LIN {X 0,Y 420.227,Z 348.89,A -85,B 0,C 180,E1 -10155.703,E2 -10155.703} C_VEL
LIN {X 0,Y 419.508,Z 359.488,A -85,B 0,C 180,E1 -10156.806,E2 -10156.806} C_VEL
LIN {X 0,Y 418.942,Z 368.019,A -85,B 0,C 180,E1 -10157.896,E2 -10157.896} C_VEL
LIN {X 0,Y 418.299,Z 375.888,A -85,B 0,C 180,E1 -10159.105,E2 -10159.105} C_VEL
LIN {X 0,Y 417.781,Z 383.575,A -85,B 0,C 180,E1 -10160.56,E2 -10160.56} C_VEL
LIN {X 0,Y 417.366,Z 390.664,A -85,B 0,C 180,E1 -10162.258,E2 -10162.258} C_VEL
LIN {X 0,Y 417.141,Z 395.456,A -85,B 0,C 180,E1 -10163.739,E2 -10163.739} C_VEL
LIN {X 0,Y 417.106,Z 398.985,A -85,B 0,C 180,E1 -10165.167,E2 -10165.167} C_VEL
LIN {X 0,Y 416.998,Z 400.842,A -85,B 0,C 180,E1 -10166.135,E2 -10166.135} C_VEL
LIN {X 0,Y 417.018,Z 402.236,A -85,B 0,C 180,E1 -10167.102,E2 -10167.102} C_VEL
LIN {X 0,Y 417.055,Z 403.232,A -85,B 0,C 180,E1 -10168.069,E2 -10168.069} C_VEL
LIN {X 0,Y 416.984,Z 404.052,A -85,B 0,C 180,E1 -10170,E2 -10170} C_VEL
LIN {X 0,Y 417.055,Z 403.229,A -85,B 0,C 180,E1 -10171.931,E2 -10171.931} C_VEL
LIN {X 0,Y 417.018,Z 402.232,A -85,B 0,C 180,E1 -10172.898,E2 -10172.898} C_VEL
LIN {X 0,Y 416.998,Z 400.835,A -85,B 0,C 180,E1 -10173.866,E2 -10173.866} C_VEL
LIN {X 0,Y 417.122,Z 397.902,A -85,B 0,C 180,E1 -10175.317,E2 -10175.317} C_VEL
LIN {X 0,Y 417.234,Z 393.93,A -85,B 0,C 180,E1 -10176.772,E2 -10176.772} C_VEL
LIN {X 0,Y 417.522,Z 387.822,A -85,B 0,C 180,E1 -10178.47,E2 -10178.47} C_VEL
LIN {X 0,Y 417.931,Z 381.149,A -85,B 0,C 180,E1 -10179.925,E2 -10179.925} C_VEL
LIN {X 0,Y 418.509,Z 372.87,A -85,B 0,C 180,E1 -10181.38,E2 -10181.38} C_VEL
LIN {X 0,Y 419.228,Z 364.386,A -85,B 0,C 180,E1 -10182.588,E2 -10182.588} C_VEL
LIN {X 0,Y 419.889,Z 353.882,A -85,B 0,C 180,E1 -10183.8,E2 -10183.8} C_VEL
LIN {X 0,Y 420.7,Z 342.093,A -85,B 0,C 180,E1 -10184.883,E2 -10184.883} C_VEL
LIN {X 0,Y 421.458,Z 330.219,A -85,B 0,C 180,E1 -10185.722,E2 -10185.722} C_VEL
LIN {X 0,Y 422.07,Z 317.862,A -85,B 0,C 180,E1 -10186.381,E2 -10186.381} C_VEL
LIN {X 0,Y 422.722,Z 305.172,A -85,B 0,C 180,E1 -10186.852,E2 -10186.852} C_VEL
LIN {X 0,Y 423.018,Z 291.859,A -85,B 0,C 180,E1 -10187.151,E2 -10187.151} C_VEL
LIN {X 0,Y 423.707,Z 215.963,A -85,B 0,C 180,E1 -10188.445,E2 -10188.445} C_VEL
LIN {X 0,Y 419.677,Z 191.543,A -85,B 0,C 180,E1 -10189.081,E2 -10189.081} C_VEL
LIN {X 0,Y 420.834,Z 174.196,A -85,B 0,C 180,E1 -10192.588,E2 -10192.588} C_VEL
LIN {X 0,Y 421.039,Z 167.944,A -85,B 0,C 180,E1 -10193.877,E2 -10193.877} C_VEL
LIN {X 0,Y 418.547,Z 155.355,A -85,B 0,C 180,E1 -10196.69,E2 -10196.69} C_VEL
LIN {X 0,Y 418.225,Z 153.888,A -85,B 0,C 180,E1 -10197.047,E2 -10197.047} C_VEL
LIN {X 0,Y 418.241,Z 153.882,A -85,B 0,C 180,E1 -10200.272,E2 -10200.272} C_VEL
LIN {X 0,Y 418.233,Z 153.885,A -85,B 0,C 180,E1 -10203.678,E2 -10203.678} C_VEL
LIN {X 0,Y 418.239,Z 153.886,A -85,B 0,C 180,E1 -10207.224,E2 -10207.224} C_VEL
LIN {X 0,Y 418.213,Z 153.892,A -85,B 0,C 180,E1 -10210.868,E2 -10210.868} C_VEL
LIN {X 0,Y 418.208,Z 153.887,A -85,B 0,C 180,E1 -10213.729,E2 -10213.729} C_VEL
LIN {X 0,Y 418.208,Z 153.894,A -85,B 0,C 180,E1 -10216.448,E2 -10216.448} C_VEL
LIN {X 0,Y 418.22,Z 153.886,A -85,B 0,C 180,E1 -10219.13,E2 -10219.13} C_VEL
LIN {X 0,Y 418.224,Z 153.89,A -85,B 0,C 180,E1 -10222.167,E2 -10222.167} C_VEL
LIN {X 0,Y 418.265,Z 153.88,A -85,B 0,C 180,E1 -10225.42,E2 -10225.42} C_VEL
LIN {X 0,Y 418.211,Z 153.889,A -85,B 0,C 180,E1 -10228.604,E2 -10228.604} C_VEL
LIN {X 0,Y 418.248,Z 153.888,A -85,B 0,C 180,E1 -10231.933,E2 -10231.933} C_VEL
LIN {X 0,Y 418.271,Z 153.88,A -85,B 0,C 180,E1 -10235.161,E2 -10235.161} C_VEL
LIN {X 0,Y 418.233,Z 153.887,A -85,B 0,C 180,E1 -10238.304,E2 -10238.304} C_VEL
LIN {X 0,Y 418.28,Z 153.881,A -85,B 0,C 180,E1 -10241.383,E2 -10241.383} C_VEL
LIN {X 0,Y 418.301,Z 153.876,A -85,B 0,C 180,E1 -10244.406,E2 -10244.406} C_VEL
LIN {X 0,Y 418.355,Z 153.873,A -85,B 0,C 180,E1 -10247.386,E2 -10247.386} C_VEL
LIN {X 0,Y 418.4,Z 153.868,A -85,B 0,C 180,E1 -10251.305,E2 -10251.305} C_VEL
LIN {X 0,Y 418.509,Z 153.85,A -85,B 0,C 180,E1 -10254.217,E2 -10254.217} C_VEL
LIN {X 0,Y 418.544,Z 153.846,A -85,B 0,C 180,E1 -10258.076,E2 -10258.076} C_VEL
LIN {X 0,Y 418.671,Z 153.83,A -85,B 0,C 180,E1 -10260,E2 -10260} C_VEL
LIN {X 0,Y 418.51,Z 153.854,A -85,B 0,C 180,E1 -10262.888,E2 -10262.888} C_VEL
LIN {X 0,Y 418.461,Z 153.857,A -85,B 0,C 180,E1 -10266.516,E2 -10266.516} C_VEL
LIN {X 0,Y 418.396,Z 153.868,A -85,B 0,C 180,E1 -10268.695,E2 -10268.695} C_VEL
LIN {X 0,Y 418.315,Z 153.874,A -85,B 0,C 180,E1 -10271.631,E2 -10271.631} C_VEL
LIN {X 0,Y 418.303,Z 153.88,A -85,B 0,C 180,E1 -10274.597,E2 -10274.597} C_VEL
LIN {X 0,Y 418.288,Z 153.877,A -85,B 0,C 180,E1 -10277.604,E2 -10277.604} C_VEL
LIN {X 0,Y 418.25,Z 153.889,A -85,B 0,C 180,E1 -10280.663,E2 -10280.663} C_VEL
LIN {X 0,Y 418.288,Z 153.878,A -85,B 0,C 180,E1 -10283.781,E2 -10283.781} C_VEL
LIN {X 0,Y 418.31,Z 153.875,A -85,B 0,C 180,E1 -10287.071,E2 -10287.071} C_VEL
LIN {X 0,Y 418.245,Z 153.889,A -85,B 0,C 180,E1 -10290.272,E2 -10290.272} C_VEL
LIN {X 0,Y 418.249,Z 153.884,A -85,B 0,C 180,E1 -10293.677,E2 -10293.677} C_VEL
LIN {X 0,Y 418.24,Z 153.883,A -85,B 0,C 180,E1 -10297.224,E2 -10297.224} C_VEL
LIN {X 0,Y 418.249,Z 153.885,A -85,B 0,C 180,E1 -10299.682,E2 -10299.682} C_VEL
LIN {X 0,Y 418.231,Z 153.888,A -85,B 0,C 180,E1 -10302.321,E2 -10302.321} C_VEL
LIN {X 0,Y 418.238,Z 153.884,A -85,B 0,C 180,E1 -10305.109,E2 -10305.109} C_VEL
LIN {X 0,Y 418.241,Z 153.89,A -85,B 0,C 180,E1 -10307.767,E2 -10307.767} C_VEL
LIN {X 0,Y 418.246,Z 153.882,A -85,B 0,C 180,E1 -10310.621,E2 -10310.621} C_VEL
LIN {X 0,Y 418.244,Z 153.886,A -85,B 0,C 180,E1 -10313.976,E2 -10313.976} C_VEL
LIN {X 0,Y 418.258,Z 153.884,A -85,B 0,C 180,E1 -10317.156,E2 -10317.156} C_VEL
LIN {X 0,Y 418.27,Z 153.881,A -85,B 0,C 180,E1 -10320.896,E2 -10320.896} C_VEL
LIN {X 0,Y 418.273,Z 153.883,A -85,B 0,C 180,E1 -10324.096,E2 -10324.096} C_VEL
LIN {X 0,Y 418.313,Z 154.005,A -85,B 0,C 180,E1 -10326.418,E2 -10326.418} C_VEL
LIN {X 0,Y 420.295,Z 164.49,A -85,B 0,C 180,E1 -10328.93,E2 -10328.93} C_VEL
LIN {X 0,Y 419.968,Z 173.899,A -85,B 0,C 180,E1 -10331.005,E2 -10331.005} C_VEL
LIN {X 0,Y 424.02,Z 194.652,A -85,B 0,C 180,E1 -10331.563,E2 -10331.563} C_VEL
LIN {X 0,Y 423.016,Z 281.721,A -85,B 0,C 180,E1 -10333.066,E2 -10333.066} C_VEL
LIN {X 0,Y 422.575,Z 295.567,A -85,B 0,C 180,E1 -10333.515,E2 -10333.515} C_VEL
LIN {X 0,Y 422.004,Z 307.965,A -85,B 0,C 180,E1 -10334.113,E2 -10334.113} C_VEL
LIN {X 0,Y 421.353,Z 319.817,A -85,B 0,C 180,E1 -10334.893,E2 -10334.893} C_VEL
LIN {X 0,Y 420.63,Z 331.686,A -85,B 0,C 180,E1 -10335.904,E2 -10335.904} C_VEL
LIN {X 0,Y 420.036,Z 341.425,A -85,B 0,C 180,E1 -10336.945,E2 -10336.945} C_VEL
LIN {X 0,Y 419.255,Z 350.619,A -85,B 0,C 180,E1 -10338.15,E2 -10338.15} C_VEL
LIN {X 0,Y 418.86,Z 356.231,A -85,B 0,C 180,E1 -10339.025,E2 -10339.025} C_VEL
LIN {X 0,Y 417.873,Z 359.92,A -85,B 0,C 180,E1 -10339.644,E2 -10339.644} C_VEL
LIN {X 0,Y 414.573,Z 365.473,A -85,B 0,C 180,E1 -10340.681,E2 -10340.681} C_VEL
LIN {X 0,Y 411.373,Z 370.436,A -85,B 0,C 180,E1 -10341.792,E2 -10341.792} C_VEL
LIN {X 0,Y 410.551,Z 373.07,A -85,B 0,C 180,E1 -10342.518,E2 -10342.518} C_VEL
LIN {X 0,Y 410.317,Z 377.758,A -85,B 0,C 180,E1 -10344.101,E2 -10344.101} C_VEL
LIN {X 0,Y 410.161,Z 380.048,A -85,B 0,C 180,E1 -10345.085,E2 -10345.085} C_VEL
LIN {X 0,Y 410.046,Z 381.911,A -85,B 0,C 180,E1 -10346.069,E2 -10346.069} C_VEL
LIN {X 0,Y 410.046,Z 383.313,A -85,B 0,C 180,E1 -10347.053,E2 -10347.053} C_VEL
LIN {X 0,Y 410.014,Z 384.31,A -85,B 0,C 180,E1 -10348.035,E2 -10348.035} C_VEL
LIN {X 0,Y 409.909,Z 385.161,A -85,B 0,C 180,E1 -10350,E2 -10350} C_VEL
LIN {X 0,Y 409.94,Z 384.973,A -85,B 0,C 180,E1 -10350.982,E2 -10350.982} C_VEL
LIN {X 0,Y 410.014,Z 384.387,A -85,B 0,C 180,E1 -10351.965,E2 -10351.965} C_VEL
LIN {X 0,Y 410.045,Z 383.42,A -85,B 0,C 180,E1 -10352.947,E2 -10352.947} C_VEL
LIN {X 0,Y 410.04,Z 382.065,A -85,B 0,C 180,E1 -10353.931,E2 -10353.931} C_VEL
LIN {X 0,Y 410.255,Z 379.195,A -85,B 0,C 180,E1 -10355.406,E2 -10355.406} C_VEL
LIN {X 0,Y 410.429,Z 375.307,A -85,B 0,C 180,E1 -10356.884,E2 -10356.884} C_VEL
LIN {X 0,Y 410.753,Z 370.29,A -85,B 0,C 180,E1 -10358.362,E2 -10358.362} C_VEL
LIN {X 0,Y 411.288,Z 363.973,A -85,B 0,C 180,E1 -10359.839,E2 -10359.839} C_VEL
LIN {X 0,Y 411.856,Z 356.067,A -85,B 0,C 180,E1 -10361.317,E2 -10361.317} C_VEL
LIN {X 0,Y 412.563,Z 348.005,A -85,B 0,C 180,E1 -10362.544,E2 -10362.544} C_VEL
LIN {X 0,Y 413.371,Z 338.166,A -85,B 0,C 180,E1 -10363.77,E2 -10363.77} C_VEL
LIN {X 0,Y 413.993,Z 328.489,A -85,B 0,C 180,E1 -10364.752,E2 -10364.752} C_VEL
LIN {X 0,Y 414.652,Z 318.019,A -85,B 0,C 180,E1 -10365.609,E2 -10365.609} C_VEL
LIN {X 0,Y 415.39,Z 305.406,A -85,B 0,C 180,E1 -10366.4,E2 -10366.4} C_VEL
LIN {X 0,Y 415.927,Z 292.786,A -85,B 0,C 180,E1 -10366.978,E2 -10366.978} C_VEL
LIN {X 0,Y 416.33,Z 280.841,A -85,B 0,C 180,E1 -10367.341,E2 -10367.341} C_VEL
LIN {X 0,Y 417.233,Z 195.021,A -85,B 0,C 180,E1 -10368.844,E2 -10368.844} C_VEL
LIN {X 0,Y 413.083,Z 173.984,A -85,B 0,C 180,E1 -10369.44,E2 -10369.44} C_VEL
LIN {X 0,Y 413.428,Z 166.217,A -85,B 0,C 180,E1 -10371.176,E2 -10371.176} C_VEL
LIN {X 0,Y 411.278,Z 154.753,A -85,B 0,C 180,E1 -10374.011,E2 -10374.011} C_VEL
LIN {X 0,Y 411.261,Z 154.753,A -85,B 0,C 180,E1 -10377.477,E2 -10377.477} C_VEL
LIN {X 0,Y 411.191,Z 154.766,A -85,B 0,C 180,E1 -10380.847,E2 -10380.847} C_VEL
LIN {X 0,Y 411.206,Z 154.764,A -85,B 0,C 180,E1 -10384.333,E2 -10384.333} C_VEL
LIN {X 0,Y 411.192,Z 154.764,A -85,B 0,C 180,E1 -10387.974,E2 -10387.974} C_VEL
LIN {X 0,Y 411.164,Z 154.765,A -85,B 0,C 180,E1 -10391.228,E2 -10391.228} C_VEL
LIN {X 0,Y 411.177,Z 154.767,A -85,B 0,C 180,E1 -10394.49,E2 -10394.49} C_VEL
LIN {X 0,Y 411.178,Z 154.769,A -85,B 0,C 180,E1 -10398.194,E2 -10398.194} C_VEL
LIN {X 0,Y 411.217,Z 154.758,A -85,B 0,C 180,E1 -10400.776,E2 -10400.776} C_VEL
LIN {X 0,Y 411.198,Z 154.762,A -85,B 0,C 180,E1 -10404.471,E2 -10404.471} C_VEL
LIN {X 0,Y 411.207,Z 154.759,A -85,B 0,C 180,E1 -10406.873,E2 -10406.873} C_VEL
LIN {X 0,Y 411.232,Z 154.756,A -85,B 0,C 180,E1 -10410.644,E2 -10410.644} C_VEL
LIN {X 0,Y 411.237,Z 154.763,A -85,B 0,C 180,E1 -10413.619,E2 -10413.619} C_VEL
LIN {X 0,Y 411.203,Z 154.761,A -85,B 0,C 180,E1 -10416.852,E2 -10416.852} C_VEL
LIN {X 0,Y 411.215,Z 154.759,A -85,B 0,C 180,E1 -10420.05,E2 -10420.05} C_VEL
LIN {X 0,Y 411.262,Z 154.757,A -85,B 0,C 180,E1 -10423.131,E2 -10423.131} C_VEL
LIN {X 0,Y 411.305,Z 154.751,A -85,B 0,C 180,E1 -10426.896,E2 -10426.896} C_VEL
LIN {X 0,Y 411.292,Z 154.749,A -85,B 0,C 180,E1 -10430.161,E2 -10430.161} C_VEL
LIN {X 0,Y 411.451,Z 154.735,A -85,B 0,C 180,E1 -10433.133,E2 -10433.133} C_VEL
LIN {X 0,Y 411.309,Z 154.752,A -85,B 0,C 180,E1 -10435.099,E2 -10435.099} C_VEL
LIN {X 0,Y 411.513,Z 154.721,A -85,B 0,C 180,E1 -10438.043,E2 -10438.043} C_VEL
LIN {X 0,Y 411.639,Z 154.706,A -85,B 0,C 180,E1 -10440,E2 -10440} C_VEL
LIN {X 0,Y 411.464,Z 154.732,A -85,B 0,C 180,E1 -10442.937,E2 -10442.937} C_VEL
LIN {X 0,Y 411.451,Z 154.733,A -85,B 0,C 180,E1 -10446.867,E2 -10446.867} C_VEL
LIN {X 0,Y 411.291,Z 154.75,A -85,B 0,C 180,E1 -10449.839,E2 -10449.839} C_VEL
LIN {X 0,Y 411.304,Z 154.748,A -85,B 0,C 180,E1 -10453.104,E2 -10453.104} C_VEL
LIN {X 0,Y 411.256,Z 154.754,A -85,B 0,C 180,E1 -10456.889,E2 -10456.889} C_VEL
LIN {X 0,Y 411.23,Z 154.761,A -85,B 0,C 180,E1 -10459.987,E2 -10459.987} C_VEL
LIN {X 0,Y 411.195,Z 154.761,A -85,B 0,C 180,E1 -10463.148,E2 -10463.148} C_VEL
LIN {X 0,Y 411.236,Z 154.759,A -85,B 0,C 180,E1 -10466.381,E2 -10466.381} C_VEL
LIN {X 0,Y 411.2,Z 154.765,A -85,B 0,C 180,E1 -10469.713,E2 -10469.713} C_VEL
LIN {X 0,Y 411.206,Z 154.76,A -85,B 0,C 180,E1 -10473.156,E2 -10473.156} C_VEL
LIN {X 0,Y 411.191,Z 154.762,A -85,B 0,C 180,E1 -10476.553,E2 -10476.553} C_VEL
LIN {X 0,Y 411.206,Z 154.765,A -85,B 0,C 180,E1 -10479.727,E2 -10479.727} C_VEL
LIN {X 0,Y 411.17,Z 154.767,A -85,B 0,C 180,E1 -10483.134,E2 -10483.134} C_VEL
LIN {X 0,Y 411.166,Z 154.767,A -85,B 0,C 180,E1 -10485.881,E2 -10485.881} C_VEL
LIN {X 0,Y 411.154,Z 154.767,A -85,B 0,C 180,E1 -10488.773,E2 -10488.773} C_VEL
LIN {X 0,Y 411.188,Z 154.762,A -85,B 0,C 180,E1 -10492.026,E2 -10492.026} C_VEL
LIN {X 0,Y 411.205,Z 154.761,A -85,B 0,C 180,E1 -10495.667,E2 -10495.667} C_VEL
LIN {X 0,Y 411.189,Z 154.769,A -85,B 0,C 180,E1 -10499.153,E2 -10499.153} C_VEL
LIN {X 0,Y 411.18,Z 154.765,A -85,B 0,C 180,E1 -10501.407,E2 -10501.407} C_VEL
LIN {X 0,Y 411.189,Z 154.897,A -85,B 0,C 180,E1 -10502.72,E2 -10502.72} C_VEL
LIN {X 0,Y 413.598,Z 166.561,A -85,B 0,C 180,E1 -10505.398,E2 -10505.398} C_VEL
LIN {X 0,Y 414.152,Z 171.118,A -85,B 0,C 180,E1 -10506.4,E2 -10506.4} C_VEL
LIN {X 0,Y 413.101,Z 187.124,A -85,B 0,C 180,E1 -10509.709,E2 -10509.709} C_VEL
LIN {X 0,Y 412.798,Z 191.373,A -85,B 0,C 180,E1 -10510.579,E2 -10510.579} C_VEL
LIN {X 0,Y 416.986,Z 216.971,A -85,B 0,C 180,E1 -10511.26,E2 -10511.26} C_VEL
LIN {X 0,Y 416.15,Z 299.691,A -85,B 0,C 180,E1 -10512.715,E2 -10512.715} C_VEL
LIN {X 0,Y 415.641,Z 312.159,A -85,B 0,C 180,E1 -10513.105,E2 -10513.105} C_VEL
LIN {X 0,Y 414.964,Z 325.061,A -85,B 0,C 180,E1 -10513.709,E2 -10513.709} C_VEL
LIN {X 0,Y 414.198,Z 337.311,A -85,B 0,C 180,E1 -10514.5,E2 -10514.5} C_VEL
LIN {X 0,Y 413.349,Z 348.727,A -85,B 0,C 180,E1 -10515.46,E2 -10515.46} C_VEL
LIN {X 0,Y 412.574,Z 359.328,A -85,B 0,C 180,E1 -10516.58,E2 -10516.58} C_VEL
LIN {X 0,Y 411.968,Z 367.858,A -85,B 0,C 180,E1 -10517.688,E2 -10517.688} C_VEL
LIN {X 0,Y 411.308,Z 375.727,A -85,B 0,C 180,E1 -10518.917,E2 -10518.917} C_VEL
LIN {X 0,Y 410.75,Z 383.414,A -85,B 0,C 180,E1 -10520.397,E2 -10520.397} C_VEL
LIN {X 0,Y 410.298,Z 390.502,A -85,B 0,C 180,E1 -10522.124,E2 -10522.124} C_VEL
LIN {X 0,Y 410.043,Z 395.707,A -85,B 0,C 180,E1 -10523.775,E2 -10523.775} C_VEL
LIN {X 0,Y 410.019,Z 398.823,A -85,B 0,C 180,E1 -10525.084,E2 -10525.084} C_VEL
LIN {X 0,Y 409.918,Z 400.68,A -85,B 0,C 180,E1 -10526.068,E2 -10526.068} C_VEL
LIN {X 0,Y 409.965,Z 403.07,A -85,B 0,C 180,E1 -10528.035,E2 -10528.035} C_VEL
LIN {X 0,Y 409.919,Z 403.676,A -85,B 0,C 180,E1 -10529.018,E2 -10529.018} C_VEL
LIN {X 0,Y 409.907,Z 403.89,A -85,B 0,C 180,E1 -10530,E2 -10530} C_VEL
LIN {X 0,Y 409.965,Z 403.066,A -85,B 0,C 180,E1 -10531.965,E2 -10531.965} C_VEL
LIN {X 0,Y 409.918,Z 400.673,A -85,B 0,C 180,E1 -10533.932,E2 -10533.932} C_VEL
LIN {X 0,Y 410.018,Z 397.739,A -85,B 0,C 180,E1 -10535.41,E2 -10535.41} C_VEL
LIN {X 0,Y 410.167,Z 393.766,A -85,B 0,C 180,E1 -10536.889,E2 -10536.889} C_VEL
LIN {X 0,Y 410.477,Z 387.658,A -85,B 0,C 180,E1 -10538.616,E2 -10538.616} C_VEL
LIN {X 0,Y 410.926,Z 380.984,A -85,B 0,C 180,E1 -10540.096,E2 -10540.096} C_VEL
LIN {X 0,Y 411.53,Z 372.705,A -85,B 0,C 180,E1 -10541.576,E2 -10541.576} C_VEL
LIN {X 0,Y 412.263,Z 364.22,A -85,B 0,C 180,E1 -10542.804,E2 -10542.804} C_VEL
LIN {X 0,Y 412.975,Z 353.461,A -85,B 0,C 180,E1 -10544.063,E2 -10544.063} C_VEL
LIN {X 0,Y 413.826,Z 341.927,A -85,B 0,C 180,E1 -10545.136,E2 -10545.136} C_VEL
LIN {X 0,Y 414.619,Z 330.052,A -85,B 0,C 180,E1 -10545.989,E2 -10545.989} C_VEL
LIN {X 0,Y 415.279,Z 317.693,A -85,B 0,C 180,E1 -10546.657,E2 -10546.657} C_VEL
LIN {X 0,Y 415.909,Z 304.999,A -85,B 0,C 180,E1 -10547.137,E2 -10547.137} C_VEL
LIN {X 0,Y 416.24,Z 291.677,A -85,B 0,C 180,E1 -10547.44,E2 -10547.44} C_VEL
LIN {X 0,Y 417.001,Z 216.913,A -85,B 0,C 180,E1 -10548.732,E2 -10548.732} C_VEL
LIN {X 0,Y 412.764,Z 191.485,A -85,B 0,C 180,E1 -10549.391,E2 -10549.391} C_VEL
LIN {X 0,Y 413.98,Z 174.03,A -85,B 0,C 180,E1 -10552.983,E2 -10552.983} C_VEL
LIN {X 0,Y 414.049,Z 169.026,A -85,B 0,C 180,E1 -10554.04,E2 -10554.04} C_VEL
LIN {X 0,Y 411.556,Z 156.514,A -85,B 0,C 180,E1 -10556.89,E2 -10556.89} C_VEL
LIN {X 0,Y 411.165,Z 154.766,A -85,B 0,C 180,E1 -10557.331,E2 -10557.331} C_VEL
LIN {X 0,Y 411.197,Z 154.759,A -85,B 0,C 180,E1 -10559.713,E2 -10559.713} C_VEL
LIN {X 0,Y 411.205,Z 154.764,A -85,B 0,C 180,E1 -10563.156,E2 -10563.156} C_VEL
LIN {X 0,Y 411.193,Z 154.765,A -85,B 0,C 180,E1 -10566.552,E2 -10566.552} C_VEL
LIN {X 0,Y 411.178,Z 154.763,A -85,B 0,C 180,E1 -10569.722,E2 -10569.722} C_VEL
LIN {X 0,Y 411.17,Z 154.766,A -85,B 0,C 180,E1 -10573.134,E2 -10573.134} C_VEL
LIN {X 0,Y 411.167,Z 154.765,A -85,B 0,C 180,E1 -10575.881,E2 -10575.881} C_VEL
LIN {X 0,Y 411.16,Z 154.769,A -85,B 0,C 180,E1 -10578.772,E2 -10578.772} C_VEL
LIN {X 0,Y 411.189,Z 154.765,A -85,B 0,C 180,E1 -10582.026,E2 -10582.026} C_VEL
LIN {X 0,Y 411.205,Z 154.761,A -85,B 0,C 180,E1 -10585.666,E2 -10585.666} C_VEL
LIN {X 0,Y 411.188,Z 154.762,A -85,B 0,C 180,E1 -10589.152,E2 -10589.152} C_VEL
LIN {X 0,Y 411.189,Z 154.764,A -85,B 0,C 180,E1 -10592.517,E2 -10592.517} C_VEL
LIN {X 0,Y 411.212,Z 154.764,A -85,B 0,C 180,E1 -10595.784,E2 -10595.784} C_VEL
LIN {X 0,Y 411.196,Z 154.761,A -85,B 0,C 180,E1 -10598.966,E2 -10598.966} C_VEL
LIN {X 0,Y 411.25,Z 154.757,A -85,B 0,C 180,E1 -10602.085,E2 -10602.085} C_VEL
LIN {X 0,Y 411.259,Z 154.754,A -85,B 0,C 180,E1 -10605.147,E2 -10605.147} C_VEL
LIN {X 0,Y 411.283,Z 154.751,A -85,B 0,C 180,E1 -10608.167,E2 -10608.167} C_VEL
LIN {X 0,Y 411.44,Z 154.731,A -85,B 0,C 180,E1 -10612.189,E2 -10612.189} C_VEL
LIN {X 0,Y 411.471,Z 154.727,A -85,B 0,C 180,E1 -10614.118,E2 -10614.118} C_VEL
LIN {X 0,Y 411.513,Z 154.722,A -85,B 0,C 180,E1 -10618.043,E2 -10618.043} C_VEL
LIN {X 0,Y 411.64,Z 154.706,A -85,B 0,C 180,E1 -10620,E2 -10620} C_VEL
LIN {X 0,Y 411.465,Z 154.732,A -85,B 0,C 180,E1 -10622.937,E2 -10622.937} C_VEL
LIN {X 0,Y 411.43,Z 154.737,A -85,B 0,C 180,E1 -10626.868,E2 -10626.868} C_VEL
LIN {X 0,Y 411.292,Z 154.749,A -85,B 0,C 180,E1 -10629.839,E2 -10629.839} C_VEL
LIN {X 0,Y 411.305,Z 154.751,A -85,B 0,C 180,E1 -10633.104,E2 -10633.104} C_VEL
LIN {X 0,Y 411.257,Z 154.758,A -85,B 0,C 180,E1 -10636.889,E2 -10636.889} C_VEL
LIN {X 0,Y 411.231,Z 154.757,A -85,B 0,C 180,E1 -10639.987,E2 -10639.987} C_VEL
LIN {X 0,Y 411.203,Z 154.761,A -85,B 0,C 180,E1 -10643.148,E2 -10643.148} C_VEL
LIN {X 0,Y 411.238,Z 154.762,A -85,B 0,C 180,E1 -10646.381,E2 -10646.381} C_VEL
LIN {X 0,Y 411.201,Z 154.761,A -85,B 0,C 180,E1 -10649.713,E2 -10649.713} C_VEL
LIN {X 0,Y 411.207,Z 154.759,A -85,B 0,C 180,E1 -10653.156,E2 -10653.156} C_VEL
LIN {X 0,Y 411.193,Z 154.764,A -85,B 0,C 180,E1 -10656.553,E2 -10656.553} C_VEL
LIN {X 0,Y 411.213,Z 154.762,A -85,B 0,C 180,E1 -10659.728,E2 -10659.728} C_VEL
LIN {X 0,Y 411.175,Z 154.764,A -85,B 0,C 180,E1 -10663.134,E2 -10663.134} C_VEL
LIN {X 0,Y 411.169,Z 154.771,A -85,B 0,C 180,E1 -10665.881,E2 -10665.881} C_VEL
LIN {X 0,Y 411.164,Z 154.765,A -85,B 0,C 180,E1 -10668.772,E2 -10668.772} C_VEL
LIN {X 0,Y 411.193,Z 154.764,A -85,B 0,C 180,E1 -10672.026,E2 -10672.026} C_VEL
LIN {X 0,Y 411.206,Z 154.765,A -85,B 0,C 180,E1 -10675.667,E2 -10675.667} C_VEL
LIN {X 0,Y 411.191,Z 154.765,A -85,B 0,C 180,E1 -10679.153,E2 -10679.153} C_VEL
LIN {X 0,Y 411.261,Z 154.754,A -85,B 0,C 180,E1 -10682.523,E2 -10682.523} C_VEL
LIN {X 0,Y 411.264,Z 154.844,A -85,B 0,C 180,E1 -10686.156,E2 -10686.156} C_VEL
LIN {X 0,Y 413.352,Z 165.781,A -85,B 0,C 180,E1 -10688.82,E2 -10688.82} C_VEL
LIN {X 0,Y 413.093,Z 174.033,A -85,B 0,C 180,E1 -10690.671,E2 -10690.671} C_VEL
LIN {X 0,Y 417.332,Z 195.92,A -85,B 0,C 180,E1 -10691.276,E2 -10691.276} C_VEL
LIN {X 0,Y 416.251,Z 281.899,A -85,B 0,C 180,E1 -10692.783,E2 -10692.783} C_VEL
LIN {X 0,Y 415.776,Z 295.741,A -85,B 0,C 180,E1 -10693.237,E2 -10693.237} C_VEL
LIN {X 0,Y 415.2,Z 308.134,A -85,B 0,C 180,E1 -10693.845,E2 -10693.845} C_VEL
LIN {X 0,Y 414.505,Z 319.985,A -85,B 0,C 180,E1 -10694.638,E2 -10694.638} C_VEL
LIN {X 0,Y 413.722,Z 331.853,A -85,B 0,C 180,E1 -10695.664,E2 -10695.664} C_VEL
LIN {X 0,Y 413.125,Z 341.591,A -85,B 0,C 180,E1 -10696.723,E2 -10696.723} C_VEL
LIN {X 0,Y 412.312,Z 350.784,A -85,B 0,C 180,E1 -10697.948,E2 -10697.948} C_VEL
LIN {X 0,Y 411.576,Z 359.707,A -85,B 0,C 180,E1 -10699.423,E2 -10699.423} C_VEL
LIN {X 0,Y 411.002,Z 366.891,A -85,B 0,C 180,E1 -10700.899,E2 -10700.899} C_VEL
LIN {X 0,Y 410.551,Z 373.07,A -85,B 0,C 180,E1 -10702.518,E2 -10702.518} C_VEL
LIN {X 0,Y 409.743,Z 375.514,A -85,B 0,C 180,E1 -10703.261,E2 -10703.261} C_VEL
LIN {X 0,Y 406.659,Z 378.949,A -85,B 0,C 180,E1 -10704.495,E2 -10704.495} C_VEL
LIN {X 0,Y 404.112,Z 381.173,A -85,B 0,C 180,E1 -10705.517,E2 -10705.517} C_VEL
LIN {X 0,Y 403.026,Z 382.552,A -85,B 0,C 180,E1 -10706.323,E2 -10706.323} C_VEL
LIN {X 0,Y 402.939,Z 382.912,A -85,B 0,C 180,E1 -10706.598,E2 -10706.598} C_VEL
LIN {X 0,Y 402.928,Z 384.472,A -85,B 0,C 180,E1 -10708.001,E2 -10708.001} C_VEL
LIN {X 0,Y 402.835,Z 385.323,A -85,B 0,C 180,E1 -10710,E2 -10710} C_VEL
LIN {X 0,Y 402.868,Z 385.134,A -85,B 0,C 180,E1 -10711,E2 -10711} C_VEL
LIN {X 0,Y 402.928,Z 384.548,A -85,B 0,C 180,E1 -10711.999,E2 -10711.999} C_VEL
LIN {X 0,Y 402.946,Z 383.582,A -85,B 0,C 180,E1 -10712.999,E2 -10712.999} C_VEL
LIN {X 0,Y 402.958,Z 382.226,A -85,B 0,C 180,E1 -10714,E2 -10714} C_VEL
LIN {X 0,Y 403.18,Z 379.357,A -85,B 0,C 180,E1 -10715.501,E2 -10715.501} C_VEL
LIN {X 0,Y 403.364,Z 375.469,A -85,B 0,C 180,E1 -10717.005,E2 -10717.005} C_VEL
LIN {X 0,Y 403.706,Z 370.451,A -85,B 0,C 180,E1 -10718.509,E2 -10718.509} C_VEL
LIN {X 0,Y 404.254,Z 364.134,A -85,B 0,C 180,E1 -10720.012,E2 -10720.012} C_VEL
LIN {X 0,Y 404.89,Z 356.226,A -85,B 0,C 180,E1 -10721.514,E2 -10721.514} C_VEL
LIN {X 0,Y 405.649,Z 348.163,A -85,B 0,C 180,E1 -10722.762,E2 -10722.762} C_VEL
LIN {X 0,Y 406.466,Z 338.325,A -85,B 0,C 180,E1 -10724.008,E2 -10724.008} C_VEL
LIN {X 0,Y 407.132,Z 328.647,A -85,B 0,C 180,E1 -10725.007,E2 -10725.007} C_VEL
LIN {X 0,Y 407.827,Z 318.175,A -85,B 0,C 180,E1 -10725.877,E2 -10725.877} C_VEL
LIN {X 0,Y 408.602,Z 305.56,A -85,B 0,C 180,E1 -10726.68,E2 -10726.68} C_VEL
LIN {X 0,Y 409.169,Z 292.936,A -85,B 0,C 180,E1 -10727.267,E2 -10727.267} C_VEL
LIN {X 0,Y 409.568,Z 280.984,A -85,B 0,C 180,E1 -10727.636,E2 -10727.636} C_VEL
LIN {X 0,Y 410.585,Z 196.294,A -85,B 0,C 180,E1 -10729.14,E2 -10729.14} C_VEL
LIN {X 0,Y 406.205,Z 174.104,A -85,B 0,C 180,E1 -10729.792,E2 -10729.792} C_VEL
LIN {X 0,Y 406.469,Z 167.513,A -85,B 0,C 180,E1 -10731.29,E2 -10731.29} C_VEL
LIN {X 0,Y 404.205,Z 155.634,A -85,B 0,C 180,E1 -10734.253,E2 -10734.253} C_VEL
LIN {X 0,Y 404.197,Z 155.633,A -85,B 0,C 180,E1 -10737.999,E2 -10737.999} C_VEL
LIN {X 0,Y 404.14,Z 155.64,A -85,B 0,C 180,E1 -10741.558,E2 -10741.558} C_VEL
LIN {X 0,Y 404.185,Z 155.636,A -85,B 0,C 180,E1 -10745.016,E2 -10745.016} C_VEL
LIN {X 0,Y 404.151,Z 155.641,A -85,B 0,C 180,E1 -10748.757,E2 -10748.757} C_VEL
LIN {X 0,Y 404.123,Z 155.643,A -85,B 0,C 180,E1 -10751.599,E2 -10751.599} C_VEL
LIN {X 0,Y 404.146,Z 155.642,A -85,B 0,C 180,E1 -10754.522,E2 -10754.522} C_VEL
LIN {X 0,Y 404.137,Z 155.64,A -85,B 0,C 180,E1 -10757.295,E2 -10757.295} C_VEL
LIN {X 0,Y 404.169,Z 155.642,A -85,B 0,C 180,E1 -10759.955,E2 -10759.955} C_VEL
LIN {X 0,Y 404.136,Z 155.64,A -85,B 0,C 180,E1 -10763.125,E2 -10763.125} C_VEL
LIN {X 0,Y 404.145,Z 155.642,A -85,B 0,C 180,E1 -10766.188,E2 -10766.188} C_VEL
LIN {X 0,Y 404.145,Z 155.646,A -85,B 0,C 180,E1 -10769.715,E2 -10769.715} C_VEL
LIN {X 0,Y 404.195,Z 155.635,A -85,B 0,C 180,E1 -10773.123,E2 -10773.123} C_VEL
LIN {X 0,Y 404.177,Z 155.639,A -85,B 0,C 180,E1 -10775.334,E2 -10775.334} C_VEL
LIN {X 0,Y 404.138,Z 155.64,A -85,B 0,C 180,E1 -10778.58,E2 -10778.58} C_VEL
LIN {X 0,Y 404.21,Z 155.634,A -85,B 0,C 180,E1 -10781.762,E2 -10781.762} C_VEL
LIN {X 0,Y 404.205,Z 155.634,A -85,B 0,C 180,E1 -10784.882,E2 -10784.882} C_VEL
LIN {X 0,Y 404.256,Z 155.626,A -85,B 0,C 180,E1 -10787.958,E2 -10787.958} C_VEL
LIN {X 0,Y 404.404,Z 155.607,A -85,B 0,C 180,E1 -10792.129,E2 -10792.129} C_VEL
LIN {X 0,Y 404.418,Z 155.605,A -85,B 0,C 180,E1 -10794.015,E2 -10794.015} C_VEL
LIN {X 0,Y 404.482,Z 155.597,A -85,B 0,C 180,E1 -10798.008,E2 -10798.008} C_VEL
LIN {X 0,Y 404.609,Z 155.582,A -85,B 0,C 180,E1 -10800,E2 -10800} C_VEL
LIN {X 0,Y 404.421,Z 155.609,A -85,B 0,C 180,E1 -10802.988,E2 -10802.988} C_VEL
LIN {X 0,Y 404.398,Z 155.61,A -85,B 0,C 180,E1 -10806.987,E2 -10806.987} C_VEL
LIN {X 0,Y 404.257,Z 155.627,A -85,B 0,C 180,E1 -10810.012,E2 -10810.012} C_VEL
LIN {X 0,Y 404.265,Z 155.624,A -85,B 0,C 180,E1 -10813.211,E2 -10813.211} C_VEL
LIN {X 0,Y 404.215,Z 155.631,A -85,B 0,C 180,E1 -10817.007,E2 -10817.007} C_VEL
LIN {X 0,Y 404.163,Z 155.642,A -85,B 0,C 180,E1 -10820.352,E2 -10820.352} C_VEL
LIN {X 0,Y 404.162,Z 155.639,A -85,B 0,C 180,E1 -10823.575,E2 -10823.575} C_VEL
LIN {X 0,Y 404.182,Z 155.638,A -85,B 0,C 180,E1 -10825.767,E2 -10825.767} C_VEL
LIN {X 0,Y 404.194,Z 155.64,A -85,B 0,C 180,E1 -10828,E2 -10828} C_VEL
LIN {X 0,Y 404.139,Z 155.644,A -85,B 0,C 180,E1 -10831.558,E2 -10831.558} C_VEL
LIN {X 0,Y 404.183,Z 155.635,A -85,B 0,C 180,E1 -10835.016,E2 -10835.016} C_VEL
LIN {X 0,Y 404.147,Z 155.639,A -85,B 0,C 180,E1 -10838.758,E2 -10838.758} C_VEL
LIN {X 0,Y 404.119,Z 155.649,A -85,B 0,C 180,E1 -10841.599,E2 -10841.599} C_VEL
LIN {X 0,Y 404.145,Z 155.639,A -85,B 0,C 180,E1 -10844.522,E2 -10844.522} C_VEL
LIN {X 0,Y 404.13,Z 155.647,A -85,B 0,C 180,E1 -10847.295,E2 -10847.295} C_VEL
LIN {X 0,Y 404.132,Z 155.642,A -85,B 0,C 180,E1 -10849.951,E2 -10849.951} C_VEL
LIN {X 0,Y 404.135,Z 155.647,A -85,B 0,C 180,E1 -10853.126,E2 -10853.126} C_VEL
LIN {X 0,Y 404.145,Z 155.639,A -85,B 0,C 180,E1 -10856.188,E2 -10856.188} C_VEL
LIN {X 0,Y 404.144,Z 155.645,A -85,B 0,C 180,E1 -10859.715,E2 -10859.715} C_VEL
LIN {X 0,Y 404.17,Z 155.776,A -85,B 0,C 180,E1 -10862.441,E2 -10862.441} C_VEL
LIN {X 0,Y 406.597,Z 167.647,A -85,B 0,C 180,E1 -10865.219,E2 -10865.219} C_VEL
LIN {X 0,Y 407.207,Z 172.486,A -85,B 0,C 180,E1 -10866.304,E2 -10866.304} C_VEL
LIN {X 0,Y 406.063,Z 188.873,A -85,B 0,C 180,E1 -10869.748,E2 -10869.748} C_VEL
LIN {X 0,Y 405.917,Z 191.21,A -85,B 0,C 180,E1 -10870.236,E2 -10870.236} C_VEL
LIN {X 0,Y 410.265,Z 217.833,A -85,B 0,C 180,E1 -10870.959,E2 -10870.959} C_VEL
LIN {X 0,Y 409.375,Z 299.542,A -85,B 0,C 180,E1 -10872.42,E2 -10872.42} C_VEL
LIN {X 0,Y 408.812,Z 312.768,A -85,B 0,C 180,E1 -10872.846,E2 -10872.846} C_VEL
LIN {X 0,Y 408.163,Z 324.905,A -85,B 0,C 180,E1 -10873.43,E2 -10873.43} C_VEL
LIN {X 0,Y 407.336,Z 337.153,A -85,B 0,C 180,E1 -10874.232,E2 -10874.232} C_VEL
LIN {X 0,Y 406.417,Z 348.995,A -85,B 0,C 180,E1 -10875.248,E2 -10875.248} C_VEL
LIN {X 0,Y 405.556,Z 360.21,A -85,B 0,C 180,E1 -10876.471,E2 -10876.471} C_VEL
LIN {X 0,Y 404.88,Z 369.374,A -85,B 0,C 180,E1 -10877.723,E2 -10877.723} C_VEL
LIN {X 0,Y 404.087,Z 378.302,A -85,B 0,C 180,E1 -10879.224,E2 -10879.224} C_VEL
LIN {X 0,Y 403.553,Z 385.489,A -85,B 0,C 180,E1 -10880.73,E2 -10880.73} C_VEL
LIN {X 0,Y 403.234,Z 390.34,A -85,B 0,C 180,E1 -10881.985,E2 -10881.985} C_VEL
LIN {X 0,Y 403.004,Z 395.2,A -85,B 0,C 180,E1 -10883.542,E2 -10883.542} C_VEL
LIN {X 0,Y 402.931,Z 398.661,A -85,B 0,C 180,E1 -10884.997,E2 -10884.997} C_VEL
LIN {X 0,Y 402.84,Z 400.518,A -85,B 0,C 180,E1 -10885.998,E2 -10885.998} C_VEL
LIN {X 0,Y 402.862,Z 402.908,A -85,B 0,C 180,E1 -10888.001,E2 -10888.001} C_VEL
LIN {X 0,Y 402.847,Z 403.514,A -85,B 0,C 180,E1 -10889,E2 -10889} C_VEL
LIN {X 0,Y 402.833,Z 403.729,A -85,B 0,C 180,E1 -10890,E2 -10890} C_VEL
LIN {X 0,Y 402.848,Z 403.511,A -85,B 0,C 180,E1 -10891,E2 -10891} C_VEL
LIN {X 0,Y 402.862,Z 402.904,A -85,B 0,C 180,E1 -10892,E2 -10892} C_VEL
LIN {X 0,Y 402.84,Z 400.51,A -85,B 0,C 180,E1 -10894.002,E2 -10894.002} C_VEL
LIN {X 0,Y 402.916,Z 397.575,A -85,B 0,C 180,E1 -10895.505,E2 -10895.505} C_VEL
LIN {X 0,Y 403.08,Z 393.602,A -85,B 0,C 180,E1 -10897.01,E2 -10897.01} C_VEL
LIN {X 0,Y 403.418,Z 387.493,A -85,B 0,C 180,E1 -10898.768,E2 -10898.768} C_VEL
LIN {X 0,Y 403.924,Z 380.82,A -85,B 0,C 180,E1 -10900.273,E2 -10900.273} C_VEL
LIN {X 0,Y 404.562,Z 372.541,A -85,B 0,C 180,E1 -10901.778,E2 -10901.778} C_VEL
LIN {X 0,Y 405.304,Z 364.055,A -85,B 0,C 180,E1 -10903.028,E2 -10903.028} C_VEL
LIN {X 0,Y 405.981,Z 354.277,A -85,B 0,C 180,E1 -10904.204,E2 -10904.204} C_VEL
LIN {X 0,Y 406.843,Z 343.189,A -85,B 0,C 180,E1 -10905.274,E2 -10905.274} C_VEL
LIN {X 0,Y 407.689,Z 331.813,A -85,B 0,C 180,E1 -10906.139,E2 -10906.139} C_VEL
LIN {X 0,Y 408.332,Z 320.127,A -85,B 0,C 180,E1 -10906.82,E2 -10906.82} C_VEL
LIN {X 0,Y 409.112,Z 306.661,A -85,B 0,C 180,E1 -10907.366,E2 -10907.366} C_VEL
LIN {X 0,Y 409.462,Z 293.285,A -85,B 0,C 180,E1 -10907.705,E2 -10907.705} C_VEL
LIN {X 0,Y 410.206,Z 217.57,A -85,B 0,C 180,E1 -10909.039,E2 -10909.039} C_VEL
LIN {X 0,Y 405.888,Z 191.318,A -85,B 0,C 180,E1 -10909.733,E2 -10909.733} C_VEL
LIN {X 0,Y 407.133,Z 173.864,A -85,B 0,C 180,E1 -10913.393,E2 -10913.393} C_VEL
LIN {X 0,Y 407.154,Z 170.652,A -85,B 0,C 180,E1 -10914.085,E2 -10914.085} C_VEL
LIN {X 0,Y 404.821,Z 158.781,A -85,B 0,C 180,E1 -10916.832,E2 -10916.832} C_VEL
LIN {X 0,Y 404.124,Z 155.642,A -85,B 0,C 180,E1 -10917.635,E2 -10917.635} C_VEL
LIN {X 0,Y 404.144,Z 155.638,A -85,B 0,C 180,E1 -10920.285,E2 -10920.285} C_VEL
LIN {X 0,Y 404.138,Z 155.64,A -85,B 0,C 180,E1 -10923.813,E2 -10923.813} C_VEL
LIN {X 0,Y 404.136,Z 155.647,A -85,B 0,C 180,E1 -10926.875,E2 -10926.875} C_VEL
LIN {X 0,Y 404.118,Z 155.643,A -85,B 0,C 180,E1 -10930.075,E2 -10930.075} C_VEL
LIN {X 0,Y 404.149,Z 155.641,A -85,B 0,C 180,E1 -10933.083,E2 -10933.083} C_VEL
LIN {X 0,Y 404.148,Z 155.64,A -85,B 0,C 180,E1 -10935.926,E2 -10935.926} C_VEL
LIN {X 0,Y 404.115,Z 155.648,A -85,B 0,C 180,E1 -10938.634,E2 -10938.634} C_VEL
LIN {X 0,Y 404.148,Z 155.639,A -85,B 0,C 180,E1 -10941.493,E2 -10941.493} C_VEL
LIN {X 0,Y 404.184,Z 155.635,A -85,B 0,C 180,E1 -10944.984,E2 -10944.984} C_VEL
LIN {X 0,Y 404.142,Z 155.642,A -85,B 0,C 180,E1 -10948.554,E2 -10948.554} C_VEL
LIN {X 0,Y 404.156,Z 155.638,A -85,B 0,C 180,E1 -10950.863,E2 -10950.863} C_VEL
LIN {X 0,Y 404.15,Z 155.643,A -85,B 0,C 180,E1 -10954.231,E2 -10954.231} C_VEL
LIN {X 0,Y 404.168,Z 155.639,A -85,B 0,C 180,E1 -10957.508,E2 -10957.508} C_VEL
LIN {X 0,Y 404.164,Z 155.637,A -85,B 0,C 180,E1 -10960.707,E2 -10960.707} C_VEL
LIN {X 0,Y 404.221,Z 155.635,A -85,B 0,C 180,E1 -10963.848,E2 -10963.848} C_VEL
LIN {X 0,Y 404.282,Z 155.623,A -85,B 0,C 180,E1 -10966.939,E2 -10966.939} C_VEL
LIN {X 0,Y 404.257,Z 155.627,A -85,B 0,C 180,E1 -10969.988,E2 -10969.988} C_VEL
LIN {X 0,Y 404.399,Z 155.61,A -85,B 0,C 180,E1 -10973.013,E2 -10973.013} C_VEL
LIN {X 0,Y 404.281,Z 155.625,A -85,B 0,C 180,E1 -10975.014,E2 -10975.014} C_VEL
LIN {X 0,Y 404.482,Z 155.598,A -85,B 0,C 180,E1 -10978.009,E2 -10978.009} C_VEL
LIN {X 0,Y 404.609,Z 155.582,A -85,B 0,C 180,E1 -10980,E2 -10980} C_VEL
LIN {X 0,Y 404.422,Z 155.61,A -85,B 0,C 180,E1 -10982.988,E2 -10982.988} C_VEL
LIN {X 0,Y 404.38,Z 155.617,A -85,B 0,C 180,E1 -10986.988,E2 -10986.988} C_VEL
LIN {X 0,Y 404.257,Z 155.625,A -85,B 0,C 180,E1 -10990.012,E2 -10990.012} C_VEL
LIN {X 0,Y 404.266,Z 155.627,A -85,B 0,C 180,E1 -10993.211,E2 -10993.211} C_VEL
LIN {X 0,Y 404.216,Z 155.634,A -85,B 0,C 180,E1 -10997.007,E2 -10997.007} C_VEL
LIN {X 0,Y 404.164,Z 155.641,A -85,B 0,C 180,E1 -11000.352,E2 -11000.352} C_VEL
LIN {X 0,Y 404.17,Z 155.636,A -85,B 0,C 180,E1 -11003.575,E2 -11003.575} C_VEL
LIN {X 0,Y 404.184,Z 155.635,A -85,B 0,C 180,E1 -11005.767,E2 -11005.767} C_VEL
LIN {X 0,Y 404.196,Z 155.635,A -85,B 0,C 180,E1 -11008,E2 -11008} C_VEL
LIN {X 0,Y 404.139,Z 155.64,A -85,B 0,C 180,E1 -11011.558,E2 -11011.558} C_VEL
LIN {X 0,Y 404.185,Z 155.634,A -85,B 0,C 180,E1 -11015.016,E2 -11015.016} C_VEL
LIN {X 0,Y 404.155,Z 155.639,A -85,B 0,C 180,E1 -11018.757,E2 -11018.757} C_VEL
LIN {X 0,Y 404.124,Z 155.644,A -85,B 0,C 180,E1 -11021.6,E2 -11021.6} C_VEL
LIN {X 0,Y 404.148,Z 155.64,A -85,B 0,C 180,E1 -11024.523,E2 -11024.523} C_VEL
LIN {X 0,Y 404.138,Z 155.642,A -85,B 0,C 180,E1 -11027.296,E2 -11027.296} C_VEL
LIN {X 0,Y 404.17,Z 155.64,A -85,B 0,C 180,E1 -11029.956,E2 -11029.956} C_VEL
LIN {X 0,Y 404.137,Z 155.642,A -85,B 0,C 180,E1 -11033.125,E2 -11033.125} C_VEL
LIN {X 0,Y 404.146,Z 155.64,A -85,B 0,C 180,E1 -11036.188,E2 -11036.188} C_VEL
LIN {X 0,Y 404.147,Z 155.643,A -85,B 0,C 180,E1 -11039.715,E2 -11039.715} C_VEL
LIN {X 0,Y 404.198,Z 155.637,A -85,B 0,C 180,E1 -11043.123,E2 -11043.123} C_VEL
LIN {X 0,Y 404.202,Z 155.689,A -85,B 0,C 180,E1 -11045.883,E2 -11045.883} C_VEL
LIN {X 0,Y 406.417,Z 167.078,A -85,B 0,C 180,E1 -11048.707,E2 -11048.707} C_VEL
LIN {X 0,Y 406.198,Z 174.187,A -85,B 0,C 180,E1 -11050.328,E2 -11050.328} C_VEL
LIN {X 0,Y 410.592,Z 196.463,A -85,B 0,C 180,E1 -11050.963,E2 -11050.963} C_VEL
LIN {X 0,Y 409.5,Z 282.077,A -85,B 0,C 180,E1 -11052.49,E2 -11052.49} C_VEL
LIN {X 0,Y 409.004,Z 295.913,A -85,B 0,C 180,E1 -11052.951,E2 -11052.951} C_VEL
LIN {X 0,Y 408.385,Z 308.304,A -85,B 0,C 180,E1 -11053.568,E2 -11053.568} C_VEL
LIN {X 0,Y 407.669,Z 320.153,A -85,B 0,C 180,E1 -11054.373,E2 -11054.373} C_VEL
LIN {X 0,Y 406.832,Z 331.977,A -85,B 0,C 180,E1 -11055.411,E2 -11055.411} C_VEL
LIN {X 0,Y 406.217,Z 341.757,A -85,B 0,C 180,E1 -11056.493,E2 -11056.493} C_VEL
LIN {X 0,Y 405.365,Z 350.949,A -85,B 0,C 180,E1 -11057.738,E2 -11057.738} C_VEL
LIN {X 0,Y 404.579,Z 359.872,A -85,B 0,C 180,E1 -11059.237,E2 -11059.237} C_VEL
LIN {X 0,Y 403.984,Z 367.055,A -85,B 0,C 180,E1 -11060.74,E2 -11060.74} C_VEL
LIN {X 0,Y 403.492,Z 373.487,A -85,B 0,C 180,E1 -11062.461,E2 -11062.461} C_VEL
LIN {X 0,Y 403.25,Z 377.922,A -85,B 0,C 180,E1 -11063.998,E2 -11063.998} C_VEL
LIN {X 0,Y 403.106,Z 380.21,A -85,B 0,C 180,E1 -11064.999,E2 -11064.999} C_VEL
LIN {X 0,Y 402.939,Z 382.912,A -85,B 0,C 180,E1 -11066.598,E2 -11066.598} C_VEL
LIN {X 0,Y 402.253,Z 383.97,A -85,B 0,C 180,E1 -11067.419,E2 -11067.419} C_VEL
LIN {X 0,Y 399.319,Z 385.062,A -85,B 0,C 180,E1 -11068.764,E2 -11068.764} C_VEL
LIN {X 0,Y 396.866,Z 385.438,A -85,B 0,C 180,E1 -11069.857,E2 -11069.857} C_VEL
LIN {X 0,Y 395.854,Z 385.388,A -85,B 0,C 180,E1 -11070.705,E2 -11070.705} C_VEL
LIN {X 0,Y 395.795,Z 385.3,A -85,B 0,C 180,E1 -11070.991,E2 -11070.991} C_VEL
LIN {X 0,Y 395.844,Z 384.71,A -85,B 0,C 180,E1 -11072.035,E2 -11072.035} C_VEL
LIN {X 0,Y 395.88,Z 382.387,A -85,B 0,C 180,E1 -11074.072,E2 -11074.072} C_VEL
LIN {X 0,Y 396.11,Z 379.518,A -85,B 0,C 180,E1 -11075.6,E2 -11075.6} C_VEL
LIN {X 0,Y 396.308,Z 375.63,A -85,B 0,C 180,E1 -11077.131,E2 -11077.131} C_VEL
LIN {X 0,Y 396.672,Z 370.612,A -85,B 0,C 180,E1 -11078.662,E2 -11078.662} C_VEL
LIN {X 0,Y 397.254,Z 364.294,A -85,B 0,C 180,E1 -11080.19,E2 -11080.19} C_VEL
LIN {X 0,Y 397.936,Z 356.386,A -85,B 0,C 180,E1 -11081.718,E2 -11081.718} C_VEL
LIN {X 0,Y 398.742,Z 348.322,A -85,B 0,C 180,E1 -11082.987,E2 -11082.987} C_VEL
LIN {X 0,Y 399.568,Z 338.483,A -85,B 0,C 180,E1 -11084.255,E2 -11084.255} C_VEL
LIN {X 0,Y 400.372,Z 327.42,A -85,B 0,C 180,E1 -11085.397,E2 -11085.397} C_VEL
LIN {X 0,Y 401.215,Z 314.809,A -85,B 0,C 180,E1 -11086.407,E2 -11086.407} C_VEL
LIN {X 0,Y 402.031,Z 302.212,A -85,B 0,C 180,E1 -11087.157,E2 -11087.157} C_VEL
LIN {X 0,Y 402.523,Z 288.677,A -85,B 0,C 180,E1 -11087.725,E2 -11087.725} C_VEL
LIN {X 0,Y 402.922,Z 276.651,A -85,B 0,C 180,E1 -11088.035,E2 -11088.035} C_VEL
LIN {X 0,Y 403.744,Z 196.484,A -85,B 0,C 180,E1 -11089.476,E2 -11089.476} C_VEL
LIN {X 0,Y 399.354,Z 174.274,A -85,B 0,C 180,E1 -11090.142,E2 -11090.142} C_VEL
LIN {X 0,Y 399.572,Z 169.612,A -85,B 0,C 180,E1 -11091.218,E2 -11091.218} C_VEL
LIN {X 0,Y 398.056,Z 161.046,A -85,B 0,C 180,E1 -11093.349,E2 -11093.349} C_VEL
LIN {X 0,Y 397.168,Z 156.511,A -85,B 0,C 180,E1 -11094.537,E2 -11094.537} C_VEL
LIN {X 0,Y 397.164,Z 156.509,A -85,B 0,C 180,E1 -11097.776,E2 -11097.776} C_VEL
LIN {X 0,Y 397.08,Z 156.523,A -85,B 0,C 180,E1 -11100.882,E2 -11100.882} C_VEL
LIN {X 0,Y 397.126,Z 156.52,A -85,B 0,C 180,E1 -11104.493,E2 -11104.493} C_VEL
LIN {X 0,Y 397.101,Z 156.522,A -85,B 0,C 180,E1 -11108.275,E2 -11108.275} C_VEL
LIN {X 0,Y 397.089,Z 156.519,A -85,B 0,C 180,E1 -11110.908,E2 -11110.908} C_VEL
LIN {X 0,Y 397.102,Z 156.518,A -85,B 0,C 180,E1 -11113.648,E2 -11113.648} C_VEL
LIN {X 0,Y 397.103,Z 156.519,A -85,B 0,C 180,E1 -11116.521,E2 -11116.521} C_VEL
LIN {X 0,Y 397.114,Z 156.518,A -85,B 0,C 180,E1 -11120.423,E2 -11120.423} C_VEL
LIN {X 0,Y 397.108,Z 156.519,A -85,B 0,C 180,E1 -11124.265,E2 -11124.265} C_VEL
LIN {X 0,Y 397.114,Z 156.515,A -85,B 0,C 180,E1 -11126.727,E2 -11126.727} C_VEL
LIN {X 0,Y 397.124,Z 156.515,A -85,B 0,C 180,E1 -11130.296,E2 -11130.296} C_VEL
LIN {X 0,Y 397.194,Z 156.505,A -85,B 0,C 180,E1 -11132.61,E2 -11132.61} C_VEL
LIN {X 0,Y 397.133,Z 156.515,A -85,B 0,C 180,E1 -11135.982,E2 -11135.982} C_VEL
LIN {X 0,Y 397.138,Z 156.516,A -85,B 0,C 180,E1 -11139.704,E2 -11139.704} C_VEL
LIN {X 0,Y 397.181,Z 156.508,A -85,B 0,C 180,E1 -11142.845,E2 -11142.845} C_VEL
LIN {X 0,Y 397.228,Z 156.502,A -85,B 0,C 180,E1 -11146.703,E2 -11146.703} C_VEL
LIN {X 0,Y 397.217,Z 156.503,A -85,B 0,C 180,E1 -11149.809,E2 -11149.809} C_VEL
LIN {X 0,Y 397.349,Z 156.491,A -85,B 0,C 180,E1 -11152.888,E2 -11152.888} C_VEL
LIN {X 0,Y 397.252,Z 156.504,A -85,B 0,C 180,E1 -11154.925,E2 -11154.925} C_VEL
LIN {X 0,Y 397.451,Z 156.473,A -85,B 0,C 180,E1 -11157.973,E2 -11157.973} C_VEL
LIN {X 0,Y 397.578,Z 156.457,A -85,B 0,C 180,E1 -11160,E2 -11160} C_VEL
LIN {X 0,Y 397.379,Z 156.485,A -85,B 0,C 180,E1 -11163.041,E2 -11163.041} C_VEL
LIN {X 0,Y 397.37,Z 156.485,A -85,B 0,C 180,E1 -11166.092,E2 -11166.092} C_VEL
LIN {X 0,Y 397.252,Z 156.499,A -85,B 0,C 180,E1 -11169.162,E2 -11169.162} C_VEL
LIN {X 0,Y 397.218,Z 156.507,A -85,B 0,C 180,E1 -11172.258,E2 -11172.258} C_VEL
LIN {X 0,Y 397.178,Z 156.507,A -85,B 0,C 180,E1 -11175.392,E2 -11175.392} C_VEL
LIN {X 0,Y 397.16,Z 156.513,A -85,B 0,C 180,E1 -11178.574,E2 -11178.574} C_VEL
LIN {X 0,Y 397.095,Z 156.521,A -85,B 0,C 180,E1 -11181.819,E2 -11181.819} C_VEL
LIN {X 0,Y 397.151,Z 156.512,A -85,B 0,C 180,E1 -11185.512,E2 -11185.512} C_VEL
LIN {X 0,Y 397.121,Z 156.515,A -85,B 0,C 180,E1 -11188.544,E2 -11188.544} C_VEL
LIN {X 0,Y 397.078,Z 156.524,A -85,B 0,C 180,E1 -11192.072,E2 -11192.072} C_VEL
LIN {X 0,Y 397.118,Z 156.519,A -85,B 0,C 180,E1 -11195.503,E2 -11195.503} C_VEL
LIN {X 0,Y 397.123,Z 156.514,A -85,B 0,C 180,E1 -11198.86,E2 -11198.86} C_VEL
LIN {X 0,Y 397.064,Z 156.522,A -85,B 0,C 180,E1 -11202.268,E2 -11202.268} C_VEL
LIN {X 0,Y 397.086,Z 156.521,A -85,B 0,C 180,E1 -11205.069,E2 -11205.069} C_VEL
LIN {X 0,Y 397.058,Z 156.523,A -85,B 0,C 180,E1 -11208.023,E2 -11208.023} C_VEL
LIN {X 0,Y 397.094,Z 156.519,A -85,B 0,C 180,E1 -11211.724,E2 -11211.724} C_VEL
LIN {X 0,Y 397.125,Z 156.516,A -85,B 0,C 180,E1 -11215.507,E2 -11215.507} C_VEL
LIN {X 0,Y 397.078,Z 156.526,A -85,B 0,C 180,E1 -11219.118,E2 -11219.118} C_VEL
LIN {X 0,Y 397.101,Z 156.552,A -85,B 0,C 180,E1 -11222.123,E2 -11222.123} C_VEL
LIN {X 0,Y 399.605,Z 168.731,A -85,B 0,C 180,E1 -11225.033,E2 -11225.033} C_VEL
LIN {X 0,Y 400.27,Z 173.75,A -85,B 0,C 180,E1 -11226.182,E2 -11226.182} C_VEL
LIN {X 0,Y 399.035,Z 190.577,A -85,B 0,C 180,E1 -11229.779,E2 -11229.779} C_VEL
LIN {X 0,Y 398.981,Z 191.122,A -85,B 0,C 180,E1 -11229.894,E2 -11229.894} C_VEL
LIN {X 0,Y 403.613,Z 219.018,A -85,B 0,C 180,E1 -11230.657,E2 -11230.657} C_VEL
LIN {X 0,Y 402.612,Z 299.392,A -85,B 0,C 180,E1 -11232.115,E2 -11232.115} C_VEL
LIN {X 0,Y 402.075,Z 311.851,A -85,B 0,C 180,E1 -11232.517,E2 -11232.517} C_VEL
LIN {X 0,Y 401.369,Z 324.749,A -85,B 0,C 180,E1 -11233.142,E2 -11233.142} C_VEL
LIN {X 0,Y 400.515,Z 336.995,A -85,B 0,C 180,E1 -11233.956,E2 -11233.956} C_VEL
LIN {X 0,Y 399.531,Z 348.836,A -85,B 0,C 180,E1 -11234.988,E2 -11234.988} C_VEL
LIN {X 0,Y 398.738,Z 359.087,A -85,B 0,C 180,E1 -11236.114,E2 -11236.114} C_VEL
LIN {X 0,Y 398.067,Z 367.538,A -85,B 0,C 180,E1 -11237.25,E2 -11237.25} C_VEL
LIN {X 0,Y 397.3,Z 375.405,A -85,B 0,C 180,E1 -11238.521,E2 -11238.521} C_VEL
LIN {X 0,Y 396.68,Z 383.091,A -85,B 0,C 180,E1 -11240.053,E2 -11240.053} C_VEL
LIN {X 0,Y 396.188,Z 390.179,A -85,B 0,C 180,E1 -11241.842,E2 -11241.842} C_VEL
LIN {X 0,Y 395.936,Z 394.896,A -85,B 0,C 180,E1 -11243.375,E2 -11243.375} C_VEL
LIN {X 0,Y 395.844,Z 398.499,A -85,B 0,C 180,E1 -11244.907,E2 -11244.907} C_VEL
LIN {X 0,Y 395.764,Z 400.357,A -85,B 0,C 180,E1 -11245.927,E2 -11245.927} C_VEL
LIN {X 0,Y 395.759,Z 402.746,A -85,B 0,C 180,E1 -11247.965,E2 -11247.965} C_VEL
LIN {X 0,Y 395.777,Z 403.353,A -85,B 0,C 180,E1 -11248.983,E2 -11248.983} C_VEL
LIN {X 0,Y 395.761,Z 403.567,A -85,B 0,C 180,E1 -11250,E2 -11250} C_VEL
LIN {X 0,Y 395.777,Z 403.35,A -85,B 0,C 180,E1 -11251.018,E2 -11251.018} C_VEL
LIN {X 0,Y 395.759,Z 402.741,A -85,B 0,C 180,E1 -11252.035,E2 -11252.035} C_VEL
LIN {X 0,Y 395.764,Z 400.348,A -85,B 0,C 180,E1 -11254.073,E2 -11254.073} C_VEL
LIN {X 0,Y 395.827,Z 396.94,A -85,B 0,C 180,E1 -11255.806,E2 -11255.806} C_VEL
LIN {X 0,Y 396.073,Z 391.844,A -85,B 0,C 180,E1 -11257.648,E2 -11257.648} C_VEL
LIN {X 0,Y 396.442,Z 386.317,A -85,B 0,C 180,E1 -11259.181,E2 -11259.181} C_VEL
LIN {X 0,Y 396.982,Z 379.419,A -85,B 0,C 180,E1 -11260.713,E2 -11260.713} C_VEL
LIN {X 0,Y 397.603,Z 372.376,A -85,B 0,C 180,E1 -11261.987,E2 -11261.987} C_VEL
LIN {X 0,Y 398.351,Z 363.889,A -85,B 0,C 180,E1 -11263.259,E2 -11263.259} C_VEL
LIN {X 0,Y 399.143,Z 353.637,A -85,B 0,C 180,E1 -11264.505,E2 -11264.505} C_VEL
LIN {X 0,Y 399.979,Z 343.023,A -85,B 0,C 180,E1 -11265.543,E2 -11265.543} C_VEL
LIN {X 0,Y 400.855,Z 331.646,A -85,B 0,C 180,E1 -11266.422,E2 -11266.422} C_VEL
LIN {X 0,Y 401.536,Z 319.957,A -85,B 0,C 180,E1 -11267.113,E2 -11267.113} C_VEL
LIN {X 0,Y 402.311,Z 306.488,A -85,B 0,C 180,E1 -11267.669,E2 -11267.669} C_VEL
LIN {X 0,Y 402.719,Z 293.104,A -85,B 0,C 180,E1 -11268.012,E2 -11268.012} C_VEL
LIN {X 0,Y 403.522,Z 218.547,A -85,B 0,C 180,E1 -11269.346,E2 -11269.346} C_VEL
LIN {X 0,Y 398.99,Z 191.151,A -85,B 0,C 180,E1 -11270.089,E2 -11270.089} C_VEL
LIN {X 0,Y 400.289,Z 173.697,A -85,B 0,C 180,E1 -11273.817,E2 -11273.817} C_VEL
LIN {X 0,Y 399.123,Z 166.296,A -85,B 0,C 180,E1 -11275.526,E2 -11275.526} C_VEL
LIN {X 0,Y 397.094,Z 156.517,A -85,B 0,C 180,E1 -11277.876,E2 -11277.876} C_VEL
LIN {X 0,Y 397.078,Z 156.525,A -85,B 0,C 180,E1 -11280.882,E2 -11280.882} C_VEL
LIN {X 0,Y 397.118,Z 156.517,A -85,B 0,C 180,E1 -11284.494,E2 -11284.494} C_VEL
LIN {X 0,Y 397.094,Z 156.519,A -85,B 0,C 180,E1 -11288.276,E2 -11288.276} C_VEL
LIN {X 0,Y 397.059,Z 156.523,A -85,B 0,C 180,E1 -11291.977,E2 -11291.977} C_VEL
LIN {X 0,Y 397.087,Z 156.52,A -85,B 0,C 180,E1 -11295.069,E2 -11295.069} C_VEL
LIN {X 0,Y 397.062,Z 156.524,A -85,B 0,C 180,E1 -11298.022,E2 -11298.022} C_VEL
LIN {X 0,Y 397.124,Z 156.514,A -85,B 0,C 180,E1 -11301.14,E2 -11301.14} C_VEL
LIN {X 0,Y 397.119,Z 156.519,A -85,B 0,C 180,E1 -11304.497,E2 -11304.497} C_VEL
LIN {X 0,Y 397.078,Z 156.523,A -85,B 0,C 180,E1 -11307.928,E2 -11307.928} C_VEL
LIN {X 0,Y 397.118,Z 156.519,A -85,B 0,C 180,E1 -11310.295,E2 -11310.295} C_VEL
LIN {X 0,Y 397.095,Z 156.521,A -85,B 0,C 180,E1 -11313.739,E2 -11313.739} C_VEL
LIN {X 0,Y 397.103,Z 156.517,A -85,B 0,C 180,E1 -11317.085,E2 -11317.085} C_VEL
LIN {X 0,Y 397.147,Z 156.512,A -85,B 0,C 180,E1 -11320.353,E2 -11320.353} C_VEL
LIN {X 0,Y 397.166,Z 156.513,A -85,B 0,C 180,E1 -11323.553,E2 -11323.553} C_VEL
LIN {X 0,Y 397.228,Z 156.501,A -85,B 0,C 180,E1 -11326.703,E2 -11326.703} C_VEL
LIN {X 0,Y 397.217,Z 156.506,A -85,B 0,C 180,E1 -11329.809,E2 -11329.809} C_VEL
LIN {X 0,Y 397.349,Z 156.487,A -85,B 0,C 180,E1 -11332.888,E2 -11332.888} C_VEL
LIN {X 0,Y 397.252,Z 156.5,A -85,B 0,C 180,E1 -11334.925,E2 -11334.925} C_VEL
LIN {X 0,Y 397.451,Z 156.474,A -85,B 0,C 180,E1 -11337.973,E2 -11337.973} C_VEL
LIN {X 0,Y 397.579,Z 156.457,A -85,B 0,C 180,E1 -11340,E2 -11340} C_VEL
LIN {X 0,Y 397.38,Z 156.488,A -85,B 0,C 180,E1 -11343.041,E2 -11343.041} C_VEL
LIN {X 0,Y 397.333,Z 156.494,A -85,B 0,C 180,E1 -11347.112,E2 -11347.112} C_VEL
LIN {X 0,Y 397.217,Z 156.503,A -85,B 0,C 180,E1 -11350.191,E2 -11350.191} C_VEL
LIN {X 0,Y 397.226,Z 156.503,A -85,B 0,C 180,E1 -11353.321,E2 -11353.321} C_VEL
LIN {X 0,Y 397.182,Z 156.509,A -85,B 0,C 180,E1 -11357.155,E2 -11357.155} C_VEL
LIN {X 0,Y 397.103,Z 156.522,A -85,B 0,C 180,E1 -11360.73,E2 -11360.73} C_VEL
LIN {X 0,Y 397.133,Z 156.514,A -85,B 0,C 180,E1 -11364.018,E2 -11364.018} C_VEL
LIN {X 0,Y 397.194,Z 156.505,A -85,B 0,C 180,E1 -11367.39,E2 -11367.39} C_VEL
LIN {X 0,Y 397.078,Z 156.521,A -85,B 0,C 180,E1 -11370.883,E2 -11370.883} C_VEL
LIN {X 0,Y 397.126,Z 156.517,A -85,B 0,C 180,E1 -11374.493,E2 -11374.493} C_VEL
LIN {X 0,Y 397.103,Z 156.521,A -85,B 0,C 180,E1 -11378.275,E2 -11378.275} C_VEL
LIN {X 0,Y 397.089,Z 156.518,A -85,B 0,C 180,E1 -11380.909,E2 -11380.909} C_VEL
LIN {X 0,Y 397.103,Z 156.52,A -85,B 0,C 180,E1 -11383.649,E2 -11383.649} C_VEL
LIN {X 0,Y 397.103,Z 156.517,A -85,B 0,C 180,E1 -11386.521,E2 -11386.521} C_VEL
LIN {X 0,Y 397.114,Z 156.516,A -85,B 0,C 180,E1 -11390.423,E2 -11390.423} C_VEL
LIN {X 0,Y 397.109,Z 156.516,A -85,B 0,C 180,E1 -11394.266,E2 -11394.266} C_VEL
LIN {X 0,Y 397.116,Z 156.515,A -85,B 0,C 180,E1 -11396.727,E2 -11396.727} C_VEL
LIN {X 0,Y 397.126,Z 156.514,A -85,B 0,C 180,E1 -11400.296,E2 -11400.296} C_VEL
LIN {X 0,Y 397.196,Z 156.507,A -85,B 0,C 180,E1 -11402.61,E2 -11402.61} C_VEL
LIN {X 0,Y 397.196,Z 156.682,A -85,B 0,C 180,E1 -11405.639,E2 -11405.639} C_VEL
LIN {X 0,Y 399.257,Z 167.235,A -85,B 0,C 180,E1 -11408.306,E2 -11408.306} C_VEL
LIN {X 0,Y 399.565,Z 169.932,A -85,B 0,C 180,E1 -11408.959,E2 -11408.959} C_VEL
LIN {X 0,Y 399.306,Z 174.354,A -85,B 0,C 180,E1 -11409.976,E2 -11409.976} C_VEL
LIN {X 0,Y 403.858,Z 197.154,A -85,B 0,C 180,E1 -11410.642,E2 -11410.642} C_VEL
LIN {X 0,Y 402.764,Z 282.255,A -85,B 0,C 180,E1 -11412.187,E2 -11412.187} C_VEL
LIN {X 0,Y 402.245,Z 296.086,A -85,B 0,C 180,E1 -11412.656,E2 -11412.656} C_VEL
LIN {X 0,Y 401.59,Z 308.473,A -85,B 0,C 180,E1 -11413.282,E2 -11413.282} C_VEL
LIN {X 0,Y 400.85,Z 320.32,A -85,B 0,C 180,E1 -11414.101,E2 -11414.101} C_VEL
LIN {X 0,Y 400.011,Z 331.475,A -85,B 0,C 180,E1 -11415.089,E2 -11415.089} C_VEL
LIN {X 0,Y 399.302,Z 341.924,A -85,B 0,C 180,E1 -11416.255,E2 -11416.255} C_VEL
LIN {X 0,Y 398.429,Z 351.114,A -85,B 0,C 180,E1 -11417.521,E2 -11417.521} C_VEL
LIN {X 0,Y 397.604,Z 360.037,A -85,B 0,C 180,E1 -11419.046,E2 -11419.046} C_VEL
LIN {X 0,Y 396.984,Z 367.219,A -85,B 0,C 180,E1 -11420.575,E2 -11420.575} C_VEL
LIN {X 0,Y 396.547,Z 372.064,A -85,B 0,C 180,E1 -11421.849,E2 -11421.849} C_VEL
LIN {X 0,Y 396.244,Z 376.66,A -85,B 0,C 180,E1 -11423.34,E2 -11423.34} C_VEL
LIN {X 0,Y 396.051,Z 380.373,A -85,B 0,C 180,E1 -11424.91,E2 -11424.91} C_VEL
LIN {X 0,Y 395.848,Z 383.147,A -85,B 0,C 180,E1 -11426.589,E2 -11426.589} C_VEL
LIN {X 0,Y 395.844,Z 384.635,A -85,B 0,C 180,E1 -11427.965,E2 -11427.965} C_VEL
LIN {X 0,Y 395.763,Z 385.484,A -85,B 0,C 180,E1 -11430,E2 -11430} C_VEL
LIN {X 0,Y 395.795,Z 385.3,A -85,B 0,C 180,E1 -11430.991,E2 -11430.991} C_VEL
LIN {X 0,Y 395.187,Z 384.981,A -85,B 0,C 180,E1 -11431.84,E2 -11431.84} C_VEL
LIN {X 0,Y 392.372,Z 383.8,A -85,B 0,C 180,E1 -11433.211,E2 -11433.211} C_VEL
LIN {X 0,Y 390.001,Z 382.28,A -85,B 0,C 180,E1 -11434.307,E2 -11434.307} C_VEL
LIN {X 0,Y 389.041,Z 380.815,A -85,B 0,C 180,E1 -11435.143,E2 -11435.143} C_VEL
LIN {X 0,Y 388.996,Z 380.247,A -85,B 0,C 180,E1 -11435.423,E2 -11435.423} C_VEL
LIN {X 0,Y 389.252,Z 375.791,A -85,B 0,C 180,E1 -11437.261,E2 -11437.261} C_VEL
LIN {X 0,Y 389.656,Z 370.773,A -85,B 0,C 180,E1 -11438.819,E2 -11438.819} C_VEL
LIN {X 0,Y 390.272,Z 364.454,A -85,B 0,C 180,E1 -11440.374,E2 -11440.374} C_VEL
LIN {X 0,Y 390.977,Z 356.546,A -85,B 0,C 180,E1 -11441.93,E2 -11441.93} C_VEL
LIN {X 0,Y 391.839,Z 348.481,A -85,B 0,C 180,E1 -11443.219,E2 -11443.219} C_VEL
LIN {X 0,Y 392.681,Z 338.642,A -85,B 0,C 180,E1 -11444.511,E2 -11444.511} C_VEL
LIN {X 0,Y 393.427,Z 328.962,A -85,B 0,C 180,E1 -11445.542,E2 -11445.542} C_VEL
LIN {X 0,Y 394.199,Z 318.487,A -85,B 0,C 180,E1 -11446.441,E2 -11446.441} C_VEL
LIN {X 0,Y 394.982,Z 306.995,A -85,B 0,C 180,E1 -11447.206,E2 -11447.206} C_VEL
LIN {X 0,Y 395.638,Z 293.999,A -85,B 0,C 180,E1 -11447.844,E2 -11447.844} C_VEL
LIN {X 0,Y 396.072,Z 282.454,A -85,B 0,C 180,E1 -11448.224,E2 -11448.224} C_VEL
LIN {X 0,Y 397.051,Z 197.43,A -85,B 0,C 180,E1 -11449.803,E2 -11449.803} C_VEL
LIN {X 0,Y 392.441,Z 174.451,A -85,B 0,C 180,E1 -11450.508,E2 -11450.508} C_VEL
LIN {X 0,Y 392.502,Z 169.533,A -85,B 0,C 180,E1 -11451.675,E2 -11451.675} C_VEL
LIN {X 0,Y 390.114,Z 157.391,A -85,B 0,C 180,E1 -11454.798,E2 -11454.798} C_VEL
LIN {X 0,Y 390.099,Z 157.39,A -85,B 0,C 180,E1 -11458.02,E2 -11458.02} C_VEL
LIN {X 0,Y 390.024,Z 157.398,A -85,B 0,C 180,E1 -11461.504,E2 -11461.504} C_VEL
LIN {X 0,Y 390.085,Z 157.391,A -85,B 0,C 180,E1 -11465.207,E2 -11465.207} C_VEL
LIN {X 0,Y 390.068,Z 157.393,A -85,B 0,C 180,E1 -11469.217,E2 -11469.217} C_VEL
LIN {X 0,Y 390.044,Z 157.401,A -85,B 0,C 180,E1 -11472.374,E2 -11472.374} C_VEL
LIN {X 0,Y 390.045,Z 157.396,A -85,B 0,C 180,E1 -11475.354,E2 -11475.354} C_VEL
LIN {X 0,Y 390.032,Z 157.403,A -85,B 0,C 180,E1 -11478.187,E2 -11478.187} C_VEL
LIN {X 0,Y 390.09,Z 157.39,A -85,B 0,C 180,E1 -11480.907,E2 -11480.907} C_VEL
LIN {X 0,Y 390.085,Z 157.391,A -85,B 0,C 180,E1 -11484.793,E2 -11484.793} C_VEL
LIN {X 0,Y 390.023,Z 157.399,A -85,B 0,C 180,E1 -11488.495,E2 -11488.495} C_VEL
LIN {X 0,Y 390.117,Z 157.389,A -85,B 0,C 180,E1 -11492.07,E2 -11492.07} C_VEL
LIN {X 0,Y 390.08,Z 157.398,A -85,B 0,C 180,E1 -11495.519,E2 -11495.519} C_VEL
LIN {X 0,Y 390.055,Z 157.396,A -85,B 0,C 180,E1 -11498.878,E2 -11498.878} C_VEL
LIN {X 0,Y 390.128,Z 157.386,A -85,B 0,C 180,E1 -11502.167,E2 -11502.167} C_VEL
LIN {X 0,Y 390.143,Z 157.389,A -85,B 0,C 180,E1 -11505.392,E2 -11505.392} C_VEL
LIN {X 0,Y 390.147,Z 157.384,A -85,B 0,C 180,E1 -11508.571,E2 -11508.571} C_VEL
LIN {X 0,Y 390.307,Z 157.363,A -85,B 0,C 180,E1 -11512.032,E2 -11512.032} C_VEL
LIN {X 0,Y 390.224,Z 157.378,A -85,B 0,C 180,E1 -11514.833,E2 -11514.833} C_VEL
LIN {X 0,Y 390.42,Z 157.349,A -85,B 0,C 180,E1 -11517.937,E2 -11517.937} C_VEL
LIN {X 0,Y 390.547,Z 157.333,A -85,B 0,C 180,E1 -11520,E2 -11520} C_VEL
LIN {X 0,Y 390.313,Z 157.365,A -85,B 0,C 180,E1 -11523.096,E2 -11523.096} C_VEL
LIN {X 0,Y 390.323,Z 157.363,A -85,B 0,C 180,E1 -11526.202,E2 -11526.202} C_VEL
LIN {X 0,Y 390.204,Z 157.376,A -85,B 0,C 180,E1 -11529.329,E2 -11529.329} C_VEL
LIN {X 0,Y 390.194,Z 157.377,A -85,B 0,C 180,E1 -11533.438,E2 -11533.438} C_VEL
LIN {X 0,Y 390.148,Z 157.383,A -85,B 0,C 180,E1 -11537.308,E2 -11537.308} C_VEL
LIN {X 0,Y 390.086,Z 157.394,A -85,B 0,C 180,E1 -11540.47,E2 -11540.47} C_VEL
LIN {X 0,Y 390.076,Z 157.394,A -85,B 0,C 180,E1 -11544.481,E2 -11544.481} C_VEL
LIN {X 0,Y 390.117,Z 157.393,A -85,B 0,C 180,E1 -11547.93,E2 -11547.93} C_VEL
LIN {X 0,Y 390.023,Z 157.401,A -85,B 0,C 180,E1 -11551.504,E2 -11551.504} C_VEL
LIN {X 0,Y 390.084,Z 157.392,A -85,B 0,C 180,E1 -11555.207,E2 -11555.207} C_VEL
LIN {X 0,Y 390.082,Z 157.393,A -85,B 0,C 180,E1 -11559.093,E2 -11559.093} C_VEL
LIN {X 0,Y 390.038,Z 157.397,A -85,B 0,C 180,E1 -11562.374,E2 -11562.374} C_VEL
LIN {X 0,Y 390.043,Z 157.402,A -85,B 0,C 180,E1 -11565.355,E2 -11565.355} C_VEL
LIN {X 0,Y 390.02,Z 157.399,A -85,B 0,C 180,E1 -11568.186,E2 -11568.186} C_VEL
LIN {X 0,Y 390.059,Z 157.397,A -85,B 0,C 180,E1 -11570.904,E2 -11570.904} C_VEL
LIN {X 0,Y 390.085,Z 157.394,A -85,B 0,C 180,E1 -11574.793,E2 -11574.793} C_VEL
LIN {X 0,Y 390.023,Z 157.4,A -85,B 0,C 180,E1 -11578.496,E2 -11578.496} C_VEL
LIN {X 0,Y 390.068,Z 157.523,A -85,B 0,C 180,E1 -11581.842,E2 -11581.842} C_VEL
LIN {X 0,Y 392.619,Z 169.816,A -85,B 0,C 180,E1 -11584.841,E2 -11584.841} C_VEL
LIN {X 0,Y 393.361,Z 174.835,A -85,B 0,C 180,E1 -11586.017,E2 -11586.017} C_VEL
LIN {X 0,Y 392.114,Z 190.996,A -85,B 0,C 180,E1 -11589.535,E2 -11589.535} C_VEL
LIN {X 0,Y 396.806,Z 218.951,A -85,B 0,C 180,E1 -11590.313,E2 -11590.313} C_VEL
LIN {X 0,Y 395.873,Z 299.243,A -85,B 0,C 180,E1 -11591.8,E2 -11591.8} C_VEL
LIN {X 0,Y 395.315,Z 311.697,A -85,B 0,C 180,E1 -11592.208,E2 -11592.208} C_VEL
LIN {X 0,Y 394.583,Z 324.593,A -85,B 0,C 180,E1 -11592.843,E2 -11592.843} C_VEL
LIN {X 0,Y 393.692,Z 336.837,A -85,B 0,C 180,E1 -11593.671,E2 -11593.671} C_VEL
LIN {X 0,Y 392.673,Z 348.42,A -85,B 0,C 180,E1 -11594.693,E2 -11594.693} C_VEL
LIN {X 0,Y 391.824,Z 359.015,A -85,B 0,C 180,E1 -11595.875,E2 -11595.875} C_VEL
LIN {X 0,Y 391.126,Z 367.378,A -85,B 0,C 180,E1 -11597.02,E2 -11597.02} C_VEL
LIN {X 0,Y 390.313,Z 375.244,A -85,B 0,C 180,E1 -11598.313,E2 -11598.313} C_VEL
LIN {X 0,Y 389.665,Z 382.93,A -85,B 0,C 180,E1 -11599.872,E2 -11599.872} C_VEL
LIN {X 0,Y 389.13,Z 390.017,A -85,B 0,C 180,E1 -11601.693,E2 -11601.693} C_VEL
LIN {X 0,Y 388.852,Z 394.733,A -85,B 0,C 180,E1 -11603.253,E2 -11603.253} C_VEL
LIN {X 0,Y 388.74,Z 398.337,A -85,B 0,C 180,E1 -11604.814,E2 -11604.814} C_VEL
LIN {X 0,Y 388.69,Z 400.195,A -85,B 0,C 180,E1 -11605.853,E2 -11605.853} C_VEL
LIN {X 0,Y 388.657,Z 402.584,A -85,B 0,C 180,E1 -11607.927,E2 -11607.927} C_VEL
LIN {X 0,Y 388.69,Z 403.191,A -85,B 0,C 180,E1 -11608.964,E2 -11608.964} C_VEL
LIN {X 0,Y 388.691,Z 403.406,A -85,B 0,C 180,E1 -11610,E2 -11610} C_VEL
LIN {X 0,Y 388.69,Z 403.188,A -85,B 0,C 180,E1 -11611.036,E2 -11611.036} C_VEL
LIN {X 0,Y 388.657,Z 402.578,A -85,B 0,C 180,E1 -11612.073,E2 -11612.073} C_VEL
LIN {X 0,Y 388.689,Z 400.185,A -85,B 0,C 180,E1 -11614.148,E2 -11614.148} C_VEL
LIN {X 0,Y 388.727,Z 397.146,A -85,B 0,C 180,E1 -11615.754,E2 -11615.754} C_VEL
LIN {X 0,Y 388.937,Z 393.275,A -85,B 0,C 180,E1 -11617.267,E2 -11617.267} C_VEL
LIN {X 0,Y 389.348,Z 387.165,A -85,B 0,C 180,E1 -11619.088,E2 -11619.088} C_VEL
LIN {X 0,Y 389.878,Z 380.491,A -85,B 0,C 180,E1 -11620.648,E2 -11620.648} C_VEL
LIN {X 0,Y 390.65,Z 372.212,A -85,B 0,C 180,E1 -11622.204,E2 -11622.204} C_VEL
LIN {X 0,Y 391.402,Z 363.723,A -85,B 0,C 180,E1 -11623.499,E2 -11623.499} C_VEL
LIN {X 0,Y 392.28,Z 353.233,A -85,B 0,C 180,E1 -11624.791,E2 -11624.791} C_VEL
LIN {X 0,Y 393.131,Z 342.856,A -85,B 0,C 180,E1 -11625.82,E2 -11625.82} C_VEL
LIN {X 0,Y 394.057,Z 331.479,A -85,B 0,C 180,E1 -11626.714,E2 -11626.714} C_VEL
LIN {X 0,Y 394.752,Z 319.788,A -85,B 0,C 180,E1 -11627.417,E2 -11627.417} C_VEL
LIN {X 0,Y 395.536,Z 306.315,A -85,B 0,C 180,E1 -11627.982,E2 -11627.982} C_VEL
LIN {X 0,Y 395.985,Z 292.923,A -85,B 0,C 180,E1 -11628.329,E2 -11628.329} C_VEL
LIN {X 0,Y 396.766,Z 218.907,A -85,B 0,C 180,E1 -11629.678,E2 -11629.678} C_VEL
LIN {X 0,Y 392.103,Z 190.983,A -85,B 0,C 180,E1 -11630.457,E2 -11630.457} C_VEL
LIN {X 0,Y 393.294,Z 176.027,A -85,B 0,C 180,E1 -11633.707,E2 -11633.707} C_VEL
LIN {X 0,Y 393.07,Z 172.272,A -85,B 0,C 180,E1 -11634.563,E2 -11634.563} C_VEL
LIN {X 0,Y 390.814,Z 160.945,A -85,B 0,C 180,E1 -11637.295,E2 -11637.295} C_VEL
LIN {X 0,Y 390.032,Z 157.395,A -85,B 0,C 180,E1 -11638.2,E2 -11638.2} C_VEL
LIN {X 0,Y 390.022,Z 157.4,A -85,B 0,C 180,E1 -11641.504,E2 -11641.504} C_VEL
LIN {X 0,Y 390.07,Z 157.395,A -85,B 0,C 180,E1 -11645.208,E2 -11645.208} C_VEL
LIN {X 0,Y 390.06,Z 157.397,A -85,B 0,C 180,E1 -11649.096,E2 -11649.096} C_VEL
LIN {X 0,Y 390.037,Z 157.4,A -85,B 0,C 180,E1 -11652.373,E2 -11652.373} C_VEL
LIN {X 0,Y 390.044,Z 157.396,A -85,B 0,C 180,E1 -11655.354,E2 -11655.354} C_VEL
LIN {X 0,Y 390.025,Z 157.402,A -85,B 0,C 180,E1 -11658.186,E2 -11658.186} C_VEL
LIN {X 0,Y 390.082,Z 157.393,A -85,B 0,C 180,E1 -11660.907,E2 -11660.907} C_VEL
LIN {X 0,Y 390.084,Z 157.392,A -85,B 0,C 180,E1 -11664.793,E2 -11664.793} C_VEL
LIN {X 0,Y 390.023,Z 157.402,A -85,B 0,C 180,E1 -11668.496,E2 -11668.496} C_VEL
LIN {X 0,Y 390.039,Z 157.403,A -85,B 0,C 180,E1 -11672.064,E2 -11672.064} C_VEL
LIN {X 0,Y 390.06,Z 157.396,A -85,B 0,C 180,E1 -11675.518,E2 -11675.518} C_VEL
LIN {X 0,Y 390.055,Z 157.394,A -85,B 0,C 180,E1 -11678.878,E2 -11678.878} C_VEL
LIN {X 0,Y 390.127,Z 157.388,A -85,B 0,C 180,E1 -11682.167,E2 -11682.167} C_VEL
LIN {X 0,Y 390.143,Z 157.387,A -85,B 0,C 180,E1 -11685.393,E2 -11685.393} C_VEL
LIN {X 0,Y 390.147,Z 157.383,A -85,B 0,C 180,E1 -11688.571,E2 -11688.571} C_VEL
LIN {X 0,Y 390.307,Z 157.364,A -85,B 0,C 180,E1 -11692.032,E2 -11692.032} C_VEL
LIN {X 0,Y 390.224,Z 157.375,A -85,B 0,C 180,E1 -11694.834,E2 -11694.834} C_VEL
LIN {X 0,Y 390.419,Z 157.35,A -85,B 0,C 180,E1 -11697.937,E2 -11697.937} C_VEL
LIN {X 0,Y 390.548,Z 157.333,A -85,B 0,C 180,E1 -11700,E2 -11700} C_VEL
LIN {X 0,Y 390.314,Z 157.368,A -85,B 0,C 180,E1 -11703.097,E2 -11703.097} C_VEL
LIN {X 0,Y 390.285,Z 157.365,A -85,B 0,C 180,E1 -11706.505,E2 -11706.505} C_VEL
LIN {X 0,Y 390.204,Z 157.379,A -85,B 0,C 180,E1 -11709.329,E2 -11709.329} C_VEL
LIN {X 0,Y 390.194,Z 157.378,A -85,B 0,C 180,E1 -11713.439,E2 -11713.439} C_VEL
LIN {X 0,Y 390.149,Z 157.384,A -85,B 0,C 180,E1 -11717.308,E2 -11717.308} C_VEL
LIN {X 0,Y 390.087,Z 157.395,A -85,B 0,C 180,E1 -11720.47,E2 -11720.47} C_VEL
LIN {X 0,Y 390.09,Z 157.39,A -85,B 0,C 180,E1 -11723.351,E2 -11723.351} C_VEL
LIN {X 0,Y 390.113,Z 157.39,A -85,B 0,C 180,E1 -11726.768,E2 -11726.768} C_VEL
LIN {X 0,Y 390.039,Z 157.403,A -85,B 0,C 180,E1 -11730.3,E2 -11730.3} C_VEL
LIN {X 0,Y 390.069,Z 157.397,A -85,B 0,C 180,E1 -11734.025,E2 -11734.025} C_VEL
LIN {X 0,Y 390.043,Z 157.397,A -85,B 0,C 180,E1 -11737.551,E2 -11737.551} C_VEL
LIN {X 0,Y 390.057,Z 157.394,A -85,B 0,C 180,E1 -11740.822,E2 -11740.822} C_VEL
LIN {X 0,Y 390.056,Z 157.401,A -85,B 0,C 180,E1 -11743.886,E2 -11743.886} C_VEL
LIN {X 0,Y 390.058,Z 157.394,A -85,B 0,C 180,E1 -11746.79,E2 -11746.79} C_VEL
LIN {X 0,Y 390.057,Z 157.399,A -85,B 0,C 180,E1 -11749.561,E2 -11749.561} C_VEL
LIN {X 0,Y 390.043,Z 157.396,A -85,B 0,C 180,E1 -11752.45,E2 -11752.45} C_VEL
LIN {X 0,Y 390.069,Z 157.394,A -85,B 0,C 180,E1 -11756.045,E2 -11756.045} C_VEL
LIN {X 0,Y 390.048,Z 157.397,A -85,B 0,C 180,E1 -11759.869,E2 -11759.869} C_VEL
LIN {X 0,Y 390.116,Z 157.392,A -85,B 0,C 180,E1 -11763.232,E2 -11763.232} C_VEL
LIN {X 0,Y 390.118,Z 157.394,A -85,B 0,C 180,E1 -11765.309,E2 -11765.309} C_VEL
LIN {X 0,Y 392.409,Z 169.145,A -85,B 0,C 180,E1 -11768.329,E2 -11768.329} C_VEL
LIN {X 0,Y 392.431,Z 174.598,A -85,B 0,C 180,E1 -11769.618,E2 -11769.618} C_VEL
LIN {X 0,Y 397.076,Z 197.66,A -85,B 0,C 180,E1 -11770.304,E2 -11770.304} C_VEL
LIN {X 0,Y 396.036,Z 282.433,A -85,B 0,C 180,E1 -11771.874,E2 -11771.874} C_VEL
LIN {X 0,Y 395.49,Z 296.258,A -85,B 0,C 180,E1 -11772.35,E2 -11772.35} C_VEL
LIN {X 0,Y 394.823,Z 308.642,A -85,B 0,C 180,E1 -11772.987,E2 -11772.987} C_VEL
LIN {X 0,Y 394.033,Z 320.488,A -85,B 0,C 180,E1 -11773.818,E2 -11773.818} C_VEL
LIN {X 0,Y 393.098,Z 332.347,A -85,B 0,C 180,E1 -11774.893,E2 -11774.893} C_VEL
LIN {X 0,Y 392.404,Z 342.09,A -85,B 0,C 180,E1 -11776.008,E2 -11776.008} C_VEL
LIN {X 0,Y 391.477,Z 351.28,A -85,B 0,C 180,E1 -11777.296,E2 -11777.296} C_VEL
LIN {X 0,Y 390.635,Z 360.202,A -85,B 0,C 180,E1 -11778.848,E2 -11778.848} C_VEL
LIN {X 0,Y 389.963,Z 367.384,A -85,B 0,C 180,E1 -11780.404,E2 -11780.404} C_VEL
LIN {X 0,Y 389.502,Z 372.229,A -85,B 0,C 180,E1 -11781.7,E2 -11781.7} C_VEL
LIN {X 0,Y 389.164,Z 377.167,A -85,B 0,C 180,E1 -11783.344,E2 -11783.344} C_VEL
LIN {X 0,Y 388.996,Z 380.536,A -85,B 0,C 180,E1 -11784.817,E2 -11784.817} C_VEL
LIN {X 0,Y 388.812,Z 382.4,A -85,B 0,C 180,E1 -11785.854,E2 -11785.854} C_VEL
LIN {X 0,Y 388.754,Z 383.801,A -85,B 0,C 180,E1 -11786.891,E2 -11786.891} C_VEL
LIN {X 0,Y 388.745,Z 384.797,A -85,B 0,C 180,E1 -11787.928,E2 -11787.928} C_VEL
LIN {X 0,Y 388.693,Z 385.646,A -85,B 0,C 180,E1 -11790,E2 -11790} C_VEL
LIN {X 0,Y 388.711,Z 385.457,A -85,B 0,C 180,E1 -11791.036,E2 -11791.036} C_VEL
LIN {X 0,Y 388.745,Z 384.872,A -85,B 0,C 180,E1 -11792.072,E2 -11792.072} C_VEL
LIN {X 0,Y 388.807,Z 382.549,A -85,B 0,C 180,E1 -11794.146,E2 -11794.146} C_VEL
LIN {X 0,Y 388.996,Z 380.247,A -85,B 0,C 180,E1 -11795.423,E2 -11795.423} C_VEL
LIN {X 0,Y 388.44,Z 378.475,A -85,B 0,C 180,E1 -11796.249,E2 -11796.249} C_VEL
LIN {X 0,Y 385.764,Z 375.158,A -85,B 0,C 180,E1 -11797.576,E2 -11797.576} C_VEL
LIN {X 0,Y 383.224,Z 371.215,A -85,B 0,C 180,E1 -11798.88,E2 -11798.88} C_VEL
LIN {X 0,Y 382.89,Z 368.389,A -85,B 0,C 180,E1 -11799.659,E2 -11799.659} C_VEL
LIN {X 0,Y 383.631,Z 360.876,A -85,B 0,C 180,E1 -11801.358,E2 -11801.358} C_VEL
LIN {X 0,Y 384.51,Z 352.055,A -85,B 0,C 180,E1 -11802.938,E2 -11802.938} C_VEL
LIN {X 0,Y 385.46,Z 343.003,A -85,B 0,C 180,E1 -11804.249,E2 -11804.249} C_VEL
LIN {X 0,Y 386.323,Z 332.438,A -85,B 0,C 180,E1 -11805.487,E2 -11805.487} C_VEL
LIN {X 0,Y 387.15,Z 321.836,A -85,B 0,C 180,E1 -11806.478,E2 -11806.478} C_VEL
LIN {X 0,Y 388.064,Z 309.322,A -85,B 0,C 180,E1 -11807.387,E2 -11807.387} C_VEL
LIN {X 0,Y 388.772,Z 296.435,A -85,B 0,C 180,E1 -11808.068,E2 -11808.068} C_VEL
LIN {X 0,Y 389.281,Z 283.74,A -85,B 0,C 180,E1 -11808.52,E2 -11808.52} C_VEL
LIN {X 0,Y 389.747,Z 253.838,A -85,B 0,C 180,E1 -11809.111,E2 -11809.111} C_VEL
LIN {X 0,Y 390.396,Z 198.498,A -85,B 0,C 180,E1 -11810.137,E2 -11810.137} C_VEL
LIN {X 0,Y 385.611,Z 174.68,A -85,B 0,C 180,E1 -11810.871,E2 -11810.871} C_VEL
LIN {X 0,Y 385.404,Z 170.071,A -85,B 0,C 180,E1 -11812.002,E2 -11812.002} C_VEL
LIN {X 0,Y 383.1,Z 158.264,A -85,B 0,C 180,E1 -11815.102,E2 -11815.102} C_VEL
LIN {X 0,Y 383.042,Z 158.272,A -85,B 0,C 180,E1 -11818.492,E2 -11818.492} C_VEL
LIN {X 0,Y 383.01,Z 158.274,A -85,B 0,C 180,E1 -11822.149,E2 -11822.149} C_VEL
LIN {X 0,Y 383.019,Z 158.276,A -85,B 0,C 180,E1 -11824.668,E2 -11824.668} C_VEL
LIN {X 0,Y 382.999,Z 158.275,A -85,B 0,C 180,E1 -11827.903,E2 -11827.903} C_VEL
LIN {X 0,Y 382.984,Z 158.275,A -85,B 0,C 180,E1 -11831.347,E2 -11831.347} C_VEL
LIN {X 0,Y 382.997,Z 158.279,A -85,B 0,C 180,E1 -11834.303,E2 -11834.303} C_VEL
LIN {X 0,Y 383.01,Z 158.272,A -85,B 0,C 180,E1 -11837.24,E2 -11837.24} C_VEL
LIN {X 0,Y 383.015,Z 158.274,A -85,B 0,C 180,E1 -11840.413,E2 -11840.413} C_VEL
LIN {X 0,Y 383.025,Z 158.275,A -85,B 0,C 180,E1 -11844.044,E2 -11844.044} C_VEL
LIN {X 0,Y 382.987,Z 158.279,A -85,B 0,C 180,E1 -11847.578,E2 -11847.578} C_VEL
LIN {X 0,Y 382.991,Z 158.276,A -85,B 0,C 180,E1 -11850.3,E2 -11850.3} C_VEL
LIN {X 0,Y 383.056,Z 158.266,A -85,B 0,C 180,E1 -11852.698,E2 -11852.698} C_VEL
LIN {X 0,Y 383.033,Z 158.27,A -85,B 0,C 180,E1 -11856.193,E2 -11856.193} C_VEL
LIN {X 0,Y 383.055,Z 158.271,A -85,B 0,C 180,E1 -11859.598,E2 -11859.598} C_VEL
LIN {X 0,Y 383.104,Z 158.263,A -85,B 0,C 180,E1 -11862.931,E2 -11862.931} C_VEL
LIN {X 0,Y 383.125,Z 158.258,A -85,B 0,C 180,E1 -11866.464,E2 -11866.464} C_VEL
LIN {X 0,Y 383.151,Z 158.255,A -85,B 0,C 180,E1 -11870.498,E2 -11870.498} C_VEL
LIN {X 0,Y 383.279,Z 158.239,A -85,B 0,C 180,E1 -11873.684,E2 -11873.684} C_VEL
LIN {X 0,Y 383.387,Z 158.225,A -85,B 0,C 180,E1 -11877.899,E2 -11877.899} C_VEL
LIN {X 0,Y 383.517,Z 158.209,A -85,B 0,C 180,E1 -11880,E2 -11880} C_VEL
LIN {X 0,Y 383.249,Z 158.244,A -85,B 0,C 180,E1 -11883.154,E2 -11883.154} C_VEL
LIN {X 0,Y 383.279,Z 158.242,A -85,B 0,C 180,E1 -11886.316,E2 -11886.316} C_VEL
LIN {X 0,Y 383.15,Z 158.255,A -85,B 0,C 180,E1 -11889.502,E2 -11889.502} C_VEL
LIN {X 0,Y 383.124,Z 158.258,A -85,B 0,C 180,E1 -11893.536,E2 -11893.536} C_VEL
LIN {X 0,Y 383.094,Z 158.262,A -85,B 0,C 180,E1 -11897.455,E2 -11897.455} C_VEL
LIN {X 0,Y 383.028,Z 158.272,A -85,B 0,C 180,E1 -11900.647,E2 -11900.647} C_VEL
LIN {X 0,Y 383.021,Z 158.274,A -85,B 0,C 180,E1 -11903.808,E2 -11903.808} C_VEL
LIN {X 0,Y 383.079,Z 158.269,A -85,B 0,C 180,E1 -11906.123,E2 -11906.123} C_VEL
LIN {X 0,Y 382.991,Z 158.279,A -85,B 0,C 180,E1 -11909.7,E2 -11909.7} C_VEL
LIN {X 0,Y 383.003,Z 158.275,A -85,B 0,C 180,E1 -11913.401,E2 -11913.401} C_VEL
LIN {X 0,Y 383.031,Z 158.271,A -85,B 0,C 180,E1 -11916.165,E2 -11916.165} C_VEL
LIN {X 0,Y 382.993,Z 158.277,A -85,B 0,C 180,E1 -11919.96,E2 -11919.96} C_VEL
LIN {X 0,Y 383.005,Z 158.273,A -85,B 0,C 180,E1 -11922.779,E2 -11922.779} C_VEL
LIN {X 0,Y 382.996,Z 158.276,A -85,B 0,C 180,E1 -11925.789,E2 -11925.789} C_VEL
LIN {X 0,Y 382.963,Z 158.279,A -85,B 0,C 180,E1 -11928.8,E2 -11928.8} C_VEL
LIN {X 0,Y 382.994,Z 158.274,A -85,B 0,C 180,E1 -11932.098,E2 -11932.098} C_VEL
LIN {X 0,Y 383.018,Z 158.275,A -85,B 0,C 180,E1 -11935.332,E2 -11935.332} C_VEL
LIN {X 0,Y 382.982,Z 158.282,A -85,B 0,C 180,E1 -11939.082,E2 -11939.082} C_VEL
LIN {X 0,Y 382.993,Z 158.312,A -85,B 0,C 180,E1 -11941.504,E2 -11941.504} C_VEL
LIN {X 0,Y 385.623,Z 170.898,A -85,B 0,C 180,E1 -11944.641,E2 -11944.641} C_VEL
LIN {X 0,Y 386.424,Z 176.21,A -85,B 0,C 180,E1 -11945.911,E2 -11945.911} C_VEL
LIN {X 0,Y 385.229,Z 190.82,A -85,B 0,C 180,E1 -11949.15,E2 -11949.15} C_VEL
LIN {X 0,Y 390.164,Z 219.974,A -85,B 0,C 180,E1 -11949.986,E2 -11949.986} C_VEL
LIN {X 0,Y 389.136,Z 299.093,A -85,B 0,C 180,E1 -11951.473,E2 -11951.473} C_VEL
LIN {X 0,Y 388.513,Z 312.306,A -85,B 0,C 180,E1 -11951.92,E2 -11951.92} C_VEL
LIN {X 0,Y 387.798,Z 324.437,A -85,B 0,C 180,E1 -11952.533,E2 -11952.533} C_VEL
LIN {X 0,Y 386.869,Z 336.679,A -85,B 0,C 180,E1 -11953.374,E2 -11953.374} C_VEL
LIN {X 0,Y 385.798,Z 348.258,A -85,B 0,C 180,E1 -11954.413,E2 -11954.413} C_VEL
LIN {X 0,Y 384.973,Z 358.194,A -85,B 0,C 180,E1 -11955.535,E2 -11955.535} C_VEL
LIN {X 0,Y 384.191,Z 367.218,A -85,B 0,C 180,E1 -11956.782,E2 -11956.782} C_VEL
LIN {X 0,Y 383.346,Z 375.084,A -85,B 0,C 180,E1 -11958.097,E2 -11958.097} C_VEL
LIN {X 0,Y 382.663,Z 382.769,A -85,B 0,C 180,E1 -11959.685,E2 -11959.685} C_VEL
LIN {X 0,Y 382.087,Z 389.856,A -85,B 0,C 180,E1 -11961.538,E2 -11961.538} C_VEL
LIN {X 0,Y 381.785,Z 394.571,A -85,B 0,C 180,E1 -11963.128,E2 -11963.128} C_VEL
LIN {X 0,Y 381.641,Z 398.175,A -85,B 0,C 180,E1 -11964.717,E2 -11964.717} C_VEL
LIN {X 0,Y 381.616,Z 400.034,A -85,B 0,C 180,E1 -11965.776,E2 -11965.776} C_VEL
LIN {X 0,Y 381.554,Z 402.421,A -85,B 0,C 180,E1 -11967.889,E2 -11967.889} C_VEL
LIN {X 0,Y 381.59,Z 403.029,A -85,B 0,C 180,E1 -11968.945,E2 -11968.945} C_VEL
LIN {X 0,Y 381.605,Z 403.244,A -85,B 0,C 180,E1 -11970,E2 -11970} C_VEL
LIN {X 0,Y 381.59,Z 403.025,A -85,B 0,C 180,E1 -11971.055,E2 -11971.055} C_VEL
LIN {X 0,Y 381.554,Z 402.416,A -85,B 0,C 180,E1 -11972.111,E2 -11972.111} C_VEL
LIN {X 0,Y 381.616,Z 400.022,A -85,B 0,C 180,E1 -11974.225,E2 -11974.225} C_VEL
LIN {X 0,Y 381.687,Z 396.385,A -85,B 0,C 180,E1 -11976.119,E2 -11976.119} C_VEL
LIN {X 0,Y 381.952,Z 391.517,A -85,B 0,C 180,E1 -11977.932,E2 -11977.932} C_VEL
LIN {X 0,Y 382.38,Z 385.989,A -85,B 0,C 180,E1 -11979.521,E2 -11979.521} C_VEL
LIN {X 0,Y 382.949,Z 379.089,A -85,B 0,C 180,E1 -11981.11,E2 -11981.11} C_VEL
LIN {X 0,Y 383.842,Z 370.459,A -85,B 0,C 180,E1 -11982.692,E2 -11982.692} C_VEL
LIN {X 0,Y 384.697,Z 360.697,A -85,B 0,C 180,E1 -11984.134,E2 -11984.134} C_VEL
LIN {X 0,Y 385.598,Z 350.713,A -85,B 0,C 180,E1 -11985.324,E2 -11985.324} C_VEL
LIN {X 0,Y 386.562,Z 339.716,A -85,B 0,C 180,E1 -11986.368,E2 -11986.368} C_VEL
LIN {X 0,Y 387.54,Z 327.39,A -85,B 0,C 180,E1 -11987.275,E2 -11987.275} C_VEL
LIN {X 0,Y 388.27,Z 315.715,A -85,B 0,C 180,E1 -11987.921,E2 -11987.921} C_VEL
LIN {X 0,Y 388.928,Z 303.26,A -85,B 0,C 180,E1 -11988.401,E2 -11988.401} C_VEL
LIN {X 0,Y 389.337,Z 287.371,A -85,B 0,C 180,E1 -11988.756,E2 -11988.756} C_VEL
LIN {X 0,Y 390.134,Z 220.067,A -85,B 0,C 180,E1 -11990.001,E2 -11990.001} C_VEL
LIN {X 0,Y 385.222,Z 190.737,A -85,B 0,C 180,E1 -11990.857,E2 -11990.857} C_VEL
LIN {X 0,Y 386.45,Z 176.158,A -85,B 0,C 180,E1 -11994.085,E2 -11994.085} C_VEL
LIN {X 0,Y 384.726,Z 166.276,A -85,B 0,C 180,E1 -11996.477,E2 -11996.477} C_VEL
LIN {X 0,Y 382.992,Z 158.272,A -85,B 0,C 180,E1 -11998.496,E2 -11998.496} C_VEL
LIN {X 0,Y 383.008,Z 158.273,A -85,B 0,C 180,E1 -12002.15,E2 -12002.15} C_VEL
LIN {X 0,Y 383.012,Z 158.276,A -85,B 0,C 180,E1 -12004.668,E2 -12004.668} C_VEL
LIN {X 0,Y 382.995,Z 158.274,A -85,B 0,C 180,E1 -12007.902,E2 -12007.902} C_VEL
LIN {X 0,Y 382.963,Z 158.279,A -85,B 0,C 180,E1 -12011.35,E2 -12011.35} C_VEL
LIN {X 0,Y 382.995,Z 158.277,A -85,B 0,C 180,E1 -12014.303,E2 -12014.303} C_VEL
LIN {X 0,Y 383.01,Z 158.272,A -85,B 0,C 180,E1 -12017.24,E2 -12017.24} C_VEL
LIN {X 0,Y 383.004,Z 158.279,A -85,B 0,C 180,E1 -12020.415,E2 -12020.415} C_VEL
LIN {X 0,Y 383.024,Z 158.274,A -85,B 0,C 180,E1 -12024.044,E2 -12024.044} C_VEL
LIN {X 0,Y 382.987,Z 158.276,A -85,B 0,C 180,E1 -12027.578,E2 -12027.578} C_VEL
LIN {X 0,Y 382.98,Z 158.28,A -85,B 0,C 180,E1 -12030.299,E2 -12030.299} C_VEL
LIN {X 0,Y 383.022,Z 158.277,A -85,B 0,C 180,E1 -12034.039,E2 -12034.039} C_VEL
LIN {X 0,Y 382.99,Z 158.276,A -85,B 0,C 180,E1 -12037.334,E2 -12037.334} C_VEL
LIN {X 0,Y 383.059,Z 158.266,A -85,B 0,C 180,E1 -12040.716,E2 -12040.716} C_VEL
LIN {X 0,Y 383.08,Z 158.266,A -85,B 0,C 180,E1 -12044.027,E2 -12044.027} C_VEL
LIN {X 0,Y 383.136,Z 158.259,A -85,B 0,C 180,E1 -12047.284,E2 -12047.284} C_VEL
LIN {X 0,Y 383.151,Z 158.254,A -85,B 0,C 180,E1 -12050.498,E2 -12050.498} C_VEL
LIN {X 0,Y 383.28,Z 158.242,A -85,B 0,C 180,E1 -12053.684,E2 -12053.684} C_VEL
LIN {X 0,Y 383.387,Z 158.226,A -85,B 0,C 180,E1 -12057.899,E2 -12057.899} C_VEL
LIN {X 0,Y 383.517,Z 158.209,A -85,B 0,C 180,E1 -12060,E2 -12060} C_VEL
LIN {X 0,Y 383.25,Z 158.249,A -85,B 0,C 180,E1 -12063.154,E2 -12063.154} C_VEL
LIN {X 0,Y 383.248,Z 158.242,A -85,B 0,C 180,E1 -12066.496,E2 -12066.496} C_VEL
LIN {X 0,Y 383.15,Z 158.256,A -85,B 0,C 180,E1 -12069.502,E2 -12069.502} C_VEL
LIN {X 0,Y 383.125,Z 158.258,A -85,B 0,C 180,E1 -12073.536,E2 -12073.536} C_VEL
LIN {X 0,Y 383.095,Z 158.262,A -85,B 0,C 180,E1 -12077.455,E2 -12077.455} C_VEL
LIN {X 0,Y 383.029,Z 158.276,A -85,B 0,C 180,E1 -12080.647,E2 -12080.647} C_VEL
LIN {X 0,Y 383.034,Z 158.27,A -85,B 0,C 180,E1 -12083.807,E2 -12083.807} C_VEL
LIN {X 0,Y 383.057,Z 158.266,A -85,B 0,C 180,E1 -12087.302,E2 -12087.302} C_VEL
LIN {X 0,Y 382.983,Z 158.276,A -85,B 0,C 180,E1 -12090.919,E2 -12090.919} C_VEL
LIN {X 0,Y 383.018,Z 158.273,A -85,B 0,C 180,E1 -12094.668,E2 -12094.668} C_VEL
LIN {X 0,Y 383,Z 158.278,A -85,B 0,C 180,E1 -12097.904,E2 -12097.904} C_VEL
LIN {X 0,Y 382.985,Z 158.276,A -85,B 0,C 180,E1 -12101.348,E2 -12101.348} C_VEL
LIN {X 0,Y 382.997,Z 158.276,A -85,B 0,C 180,E1 -12104.304,E2 -12104.304} C_VEL
LIN {X 0,Y 383.011,Z 158.273,A -85,B 0,C 180,E1 -12107.24,E2 -12107.24} C_VEL
LIN {X 0,Y 383.014,Z 158.272,A -85,B 0,C 180,E1 -12110.414,E2 -12110.414} C_VEL
LIN {X 0,Y 383.026,Z 158.272,A -85,B 0,C 180,E1 -12114.045,E2 -12114.045} C_VEL
LIN {X 0,Y 382.988,Z 158.281,A -85,B 0,C 180,E1 -12117.578,E2 -12117.578} C_VEL
LIN {X 0,Y 382.994,Z 158.274,A -85,B 0,C 180,E1 -12120.3,E2 -12120.3} C_VEL
LIN {X 0,Y 383.059,Z 158.268,A -85,B 0,C 180,E1 -12122.698,E2 -12122.698} C_VEL
LIN {X 0,Y 383.095,Z 158.398,A -85,B 0,C 180,E1 -12125.043,E2 -12125.043} C_VEL
LIN {X 0,Y 385.324,Z 169.706,A -85,B 0,C 180,E1 -12128.008,E2 -12128.008} C_VEL
LIN {X 0,Y 385.605,Z 174.467,A -85,B 0,C 180,E1 -12129.181,E2 -12129.181} C_VEL
LIN {X 0,Y 385.609,Z 174.847,A -85,B 0,C 180,E1 -12129.242,E2 -12129.242} C_VEL
LIN {X 0,Y 390.433,Z 198.643,A -85,B 0,C 180,E1 -12129.97,E2 -12129.97} C_VEL
LIN {X 0,Y 389.295,Z 281.428,A -85,B 0,C 180,E1 -12131.515,E2 -12131.515} C_VEL
LIN {X 0,Y 388.823,Z 294.909,A -85,B 0,C 180,E1 -12131.969,E2 -12131.969} C_VEL
LIN {X 0,Y 388.135,Z 307.709,A -85,B 0,C 180,E1 -12132.616,E2 -12132.616} C_VEL
LIN {X 0,Y 387.322,Z 319.069,A -85,B 0,C 180,E1 -12133.394,E2 -12133.394} C_VEL
LIN {X 0,Y 386.403,Z 330.624,A -85,B 0,C 180,E1 -12134.427,E2 -12134.427} C_VEL
LIN {X 0,Y 385.639,Z 341.195,A -85,B 0,C 180,E1 -12135.623,E2 -12135.623} C_VEL
LIN {X 0,Y 384.75,Z 349.748,A -85,B 0,C 180,E1 -12136.801,E2 -12136.801} C_VEL
LIN {X 0,Y 383.972,Z 357.626,A -85,B 0,C 180,E1 -12138.117,E2 -12138.117} C_VEL
LIN {X 0,Y 383.173,Z 365.326,A -85,B 0,C 180,E1 -12139.698,E2 -12139.698} C_VEL
LIN {X 0,Y 382.479,Z 372.392,A -85,B 0,C 180,E1 -12141.547,E2 -12141.547} C_VEL
LIN {X 0,Y 382.087,Z 377.663,A -85,B 0,C 180,E1 -12143.347,E2 -12143.347} C_VEL
LIN {X 0,Y 381.919,Z 380.699,A -85,B 0,C 180,E1 -12144.721,E2 -12144.721} C_VEL
LIN {X 0,Y 381.742,Z 382.562,A -85,B 0,C 180,E1 -12145.777,E2 -12145.777} C_VEL
LIN {X 0,Y 381.66,Z 383.964,A -85,B 0,C 180,E1 -12146.833,E2 -12146.833} C_VEL
LIN {X 0,Y 381.647,Z 384.96,A -85,B 0,C 180,E1 -12147.889,E2 -12147.889} C_VEL
LIN {X 0,Y 381.627,Z 385.574,A -85,B 0,C 180,E1 -12148.945,E2 -12148.945} C_VEL
LIN {X 0,Y 381.608,Z 385.808,A -85,B 0,C 180,E1 -12150,E2 -12150} C_VEL
LIN {X 0,Y 381.627,Z 385.619,A -85,B 0,C 180,E1 -12151.055,E2 -12151.055} C_VEL
LIN {X 0,Y 381.647,Z 385.034,A -85,B 0,C 180,E1 -12152.111,E2 -12152.111} C_VEL
LIN {X 0,Y 381.735,Z 382.71,A -85,B 0,C 180,E1 -12154.223,E2 -12154.223} C_VEL
LIN {X 0,Y 381.974,Z 379.84,A -85,B 0,C 180,E1 -12155.808,E2 -12155.808} C_VEL
LIN {X 0,Y 382.207,Z 375.952,A -85,B 0,C 180,E1 -12157.395,E2 -12157.395} C_VEL
LIN {X 0,Y 382.629,Z 370.933,A -85,B 0,C 180,E1 -12158.982,E2 -12158.982} C_VEL
LIN {X 0,Y 382.89,Z 368.389,A -85,B 0,C 180,E1 -12159.659,E2 -12159.659} C_VEL
LIN {X 0,Y 382.604,Z 365.41,A -85,B 0,C 180,E1 -12160.422,E2 -12160.422} C_VEL
LIN {X 0,Y 380.332,Z 360.225,A -85,B 0,C 180,E1 -12161.647,E2 -12161.647} C_VEL
LIN {X 0,Y 378.091,Z 354.391,A -85,B 0,C 180,E1 -12162.813,E2 -12162.813} C_VEL
LIN {X 0,Y 377.851,Z 350.394,A -85,B 0,C 180,E1 -12163.472,E2 -12163.472} C_VEL
LIN {X 0,Y 378.862,Z 340.025,A -85,B 0,C 180,E1 -12164.915,E2 -12164.915} C_VEL
LIN {X 0,Y 379.769,Z 329.277,A -85,B 0,C 180,E1 -12166.116,E2 -12166.116} C_VEL
LIN {X 0,Y 380.616,Z 318.798,A -85,B 0,C 180,E1 -12167.045,E2 -12167.045} C_VEL
LIN {X 0,Y 381.458,Z 307.303,A -85,B 0,C 180,E1 -12167.836,E2 -12167.836} C_VEL
LIN {X 0,Y 382.186,Z 294.301,A -85,B 0,C 180,E1 -12168.494,E2 -12168.494} C_VEL
LIN {X 0,Y 382.654,Z 282.745,A -85,B 0,C 180,E1 -12168.887,E2 -12168.887} C_VEL
LIN {X 0,Y 383.844,Z 200.066,A -85,B 0,C 180,E1 -12170.468,E2 -12170.468} C_VEL
LIN {X 0,Y 378.752,Z 174.868,A -85,B 0,C 180,E1 -12171.26,E2 -12171.26} C_VEL
LIN {X 0,Y 378.11,Z 169.402,A -85,B 0,C 180,E1 -12172.657,E2 -12172.657} C_VEL
LIN {X 0,Y 376.05,Z 159.143,A -85,B 0,C 180,E1 -12175.458,E2 -12175.458} C_VEL
LIN {X 0,Y 375.972,Z 159.151,A -85,B 0,C 180,E1 -12179.079,E2 -12179.079} C_VEL
LIN {X 0,Y 375.95,Z 159.155,A -85,B 0,C 180,E1 -12182.828,E2 -12182.828} C_VEL
LIN {X 0,Y 375.958,Z 159.151,A -85,B 0,C 180,E1 -12185.415,E2 -12185.415} C_VEL
LIN {X 0,Y 375.973,Z 159.154,A -85,B 0,C 180,E1 -12188.27,E2 -12188.27} C_VEL
LIN {X 0,Y 375.935,Z 159.154,A -85,B 0,C 180,E1 -12191.6,E2 -12191.6} C_VEL
LIN {X 0,Y 375.928,Z 159.154,A -85,B 0,C 180,E1 -12195.268,E2 -12195.268} C_VEL
LIN {X 0,Y 375.935,Z 159.157,A -85,B 0,C 180,E1 -12198.399,E2 -12198.399} C_VEL
LIN {X 0,Y 375.974,Z 159.152,A -85,B 0,C 180,E1 -12201.729,E2 -12201.729} C_VEL
LIN {X 0,Y 375.98,Z 159.149,A -85,B 0,C 180,E1 -12205.332,E2 -12205.332} C_VEL
LIN {X 0,Y 375.958,Z 159.151,A -85,B 0,C 180,E1 -12208.438,E2 -12208.438} C_VEL
LIN {X 0,Y 375.996,Z 159.148,A -85,B 0,C 180,E1 -12212.141,E2 -12212.141} C_VEL
LIN {X 0,Y 376.006,Z 159.145,A -85,B 0,C 180,E1 -12214.539,E2 -12214.539} C_VEL
LIN {X 0,Y 375.963,Z 159.151,A -85,B 0,C 180,E1 -12218.046,E2 -12218.046} C_VEL
LIN {X 0,Y 376.023,Z 159.148,A -85,B 0,C 180,E1 -12221.474,E2 -12221.474} C_VEL
LIN {X 0,Y 376.058,Z 159.14,A -85,B 0,C 180,E1 -12224.832,E2 -12224.832} C_VEL
LIN {X 0,Y 376.049,Z 159.139,A -85,B 0,C 180,E1 -12228.136,E2 -12228.136} C_VEL
LIN {X 0,Y 376.218,Z 159.118,A -85,B 0,C 180,E1 -12231.919,E2 -12231.919} C_VEL
LIN {X 0,Y 376.168,Z 159.127,A -85,B 0,C 180,E1 -12234.64,E2 -12234.64} C_VEL
LIN {X 0,Y 376.353,Z 159.101,A -85,B 0,C 180,E1 -12237.86,E2 -12237.86} C_VEL
LIN {X 0,Y 376.486,Z 159.085,A -85,B 0,C 180,E1 -12240,E2 -12240} C_VEL
LIN {X 0,Y 376.187,Z 159.124,A -85,B 0,C 180,E1 -12243.213,E2 -12243.213} C_VEL
LIN {X 0,Y 376.238,Z 159.12,A -85,B 0,C 180,E1 -12246.435,E2 -12246.435} C_VEL
LIN {X 0,Y 376.118,Z 159.131,A -85,B 0,C 180,E1 -12249.681,E2 -12249.681} C_VEL
LIN {X 0,Y 376.088,Z 159.135,A -85,B 0,C 180,E1 -12253.658,E2 -12253.658} C_VEL
LIN {X 0,Y 376.043,Z 159.141,A -85,B 0,C 180,E1 -12257.607,E2 -12257.607} C_VEL
LIN {X 0,Y 375.977,Z 159.149,A -85,B 0,C 180,E1 -12260.832,E2 -12260.832} C_VEL
LIN {X 0,Y 375.987,Z 159.151,A -85,B 0,C 180,E1 -12264.282,E2 -12264.282} C_VEL
LIN {X 0,Y 376.019,Z 159.144,A -85,B 0,C 180,E1 -12266.652,E2 -12266.652} C_VEL
LIN {X 0,Y 375.964,Z 159.152,A -85,B 0,C 180,E1 -12270.313,E2 -12270.313} C_VEL
LIN {X 0,Y 375.959,Z 159.153,A -85,B 0,C 180,E1 -12274.112,E2 -12274.112} C_VEL
LIN {X 0,Y 375.952,Z 159.151,A -85,B 0,C 180,E1 -12276.742,E2 -12276.742} C_VEL
LIN {X 0,Y 375.975,Z 159.151,A -85,B 0,C 180,E1 -12279.968,E2 -12279.968} C_VEL
LIN {X 0,Y 375.929,Z 159.158,A -85,B 0,C 180,E1 -12283.766,E2 -12283.766} C_VEL
LIN {X 0,Y 375.933,Z 159.155,A -85,B 0,C 180,E1 -12286.811,E2 -12286.811} C_VEL
LIN {X 0,Y 375.936,Z 159.154,A -85,B 0,C 180,E1 -12290.534,E2 -12290.534} C_VEL
LIN {X 0,Y 375.963,Z 159.153,A -85,B 0,C 180,E1 -12293.496,E2 -12293.496} C_VEL
LIN {X 0,Y 375.96,Z 159.151,A -85,B 0,C 180,E1 -12295.889,E2 -12295.889} C_VEL
LIN {X 0,Y 375.962,Z 159.157,A -85,B 0,C 180,E1 -12299.687,E2 -12299.687} C_VEL
LIN {X 0,Y 375.978,Z 159.321,A -85,B 0,C 180,E1 -12301.21,E2 -12301.21} C_VEL
LIN {X 0,Y 378.634,Z 171.981,A -85,B 0,C 180,E1 -12304.434,E2 -12304.434} C_VEL
LIN {X 0,Y 379.437,Z 176.758,A -85,B 0,C 180,E1 -12305.606,E2 -12305.606} C_VEL
LIN {X 0,Y 378.644,Z 187.097,A -85,B 0,C 180,E1 -12307.952,E2 -12307.952} C_VEL
LIN {X 0,Y 378.364,Z 190.658,A -85,B 0,C 180,E1 -12308.754,E2 -12308.754} C_VEL
LIN {X 0,Y 383.473,Z 220.778,A -85,B 0,C 180,E1 -12309.64,E2 -12309.64} C_VEL
LIN {X 0,Y 382.398,Z 298.944,A -85,B 0,C 180,E1 -12311.134,E2 -12311.134} C_VEL
LIN {X 0,Y 381.754,Z 312.152,A -85,B 0,C 180,E1 -12311.588,E2 -12311.588} C_VEL
LIN {X 0,Y 381.038,Z 324.281,A -85,B 0,C 180,E1 -12312.213,E2 -12312.213} C_VEL
LIN {X 0,Y 380.051,Z 336.521,A -85,B 0,C 180,E1 -12313.067,E2 -12313.067} C_VEL
LIN {X 0,Y 378.947,Z 348.099,A -85,B 0,C 180,E1 -12314.124,E2 -12314.124} C_VEL
LIN {X 0,Y 378.023,Z 358.754,A -85,B 0,C 180,E1 -12315.356,E2 -12315.356} C_VEL
LIN {X 0,Y 377.261,Z 367.057,A -85,B 0,C 180,E1 -12316.534,E2 -12316.534} C_VEL
LIN {X 0,Y 376.394,Z 374.923,A -85,B 0,C 180,E1 -12317.874,E2 -12317.874} C_VEL
LIN {X 0,Y 375.656,Z 382.607,A -85,B 0,C 180,E1 -12319.49,E2 -12319.49} C_VEL
LIN {X 0,Y 375.035,Z 389.694,A -85,B 0,C 180,E1 -12321.378,E2 -12321.378} C_VEL
LIN {X 0,Y 374.725,Z 394.41,A -85,B 0,C 180,E1 -12322.998,E2 -12322.998} C_VEL
LIN {X 0,Y 374.55,Z 398.013,A -85,B 0,C 180,E1 -12324.617,E2 -12324.617} C_VEL
LIN {X 0,Y 374.521,Z 399.872,A -85,B 0,C 180,E1 -12325.695,E2 -12325.695} C_VEL
LIN {X 0,Y 374.453,Z 402.259,A -85,B 0,C 180,E1 -12327.849,E2 -12327.849} C_VEL
LIN {X 0,Y 374.49,Z 402.867,A -85,B 0,C 180,E1 -12328.925,E2 -12328.925} C_VEL
LIN {X 0,Y 374.507,Z 403.082,A -85,B 0,C 180,E1 -12330,E2 -12330} C_VEL
LIN {X 0,Y 374.49,Z 402.863,A -85,B 0,C 180,E1 -12331.075,E2 -12331.075} C_VEL
LIN {X 0,Y 374.452,Z 401.256,A -85,B 0,C 180,E1 -12333.228,E2 -12333.228} C_VEL
LIN {X 0,Y 374.521,Z 399.859,A -85,B 0,C 180,E1 -12334.305,E2 -12334.305} C_VEL
LIN {X 0,Y 374.582,Z 396.613,A -85,B 0,C 180,E1 -12336.066,E2 -12336.066} C_VEL
LIN {X 0,Y 374.798,Z 392.947,A -85,B 0,C 180,E1 -12337.542,E2 -12337.542} C_VEL
LIN {X 0,Y 375.242,Z 386.836,A -85,B 0,C 180,E1 -12339.432,E2 -12339.432} C_VEL
LIN {X 0,Y 375.858,Z 380.161,A -85,B 0,C 180,E1 -12341.05,E2 -12341.05} C_VEL
LIN {X 0,Y 376.716,Z 371.882,A -85,B 0,C 180,E1 -12342.662,E2 -12342.662} C_VEL
LIN {X 0,Y 377.525,Z 363.392,A -85,B 0,C 180,E1 -12344.005,E2 -12344.005} C_VEL
LIN {X 0,Y 378.497,Z 352.901,A -85,B 0,C 180,E1 -12345.343,E2 -12345.343} C_VEL
LIN {X 0,Y 379.603,Z 341.095,A -85,B 0,C 180,E1 -12346.538,E2 -12346.538} C_VEL
LIN {X 0,Y 380.609,Z 329.213,A -85,B 0,C 180,E1 -12347.461,E2 -12347.461} C_VEL
LIN {X 0,Y 381.419,Z 316.846,A -85,B 0,C 180,E1 -12348.185,E2 -12348.185} C_VEL
LIN {X 0,Y 382.157,Z 304.136,A -85,B 0,C 180,E1 -12348.704,E2 -12348.704} C_VEL
LIN {X 0,Y 382.592,Z 290.769,A -85,B 0,C 180,E1 -12349.03,E2 -12349.03} C_VEL
LIN {X 0,Y 383.383,Z 220.255,A -85,B 0,C 180,E1 -12350.362,E2 -12350.362} C_VEL
LIN {X 0,Y 378.348,Z 190.642,A -85,B 0,C 180,E1 -12351.237,E2 -12351.237} C_VEL
LIN {X 0,Y 379.472,Z 178.188,A -85,B 0,C 180,E1 -12354.045,E2 -12354.045} C_VEL
LIN {X 0,Y 378.612,Z 171.915,A -85,B 0,C 180,E1 -12355.568,E2 -12355.568} C_VEL
LIN {X 0,Y 376.467,Z 161.602,A -85,B 0,C 180,E1 -12358.182,E2 -12358.182} C_VEL
LIN {X 0,Y 375.934,Z 159.154,A -85,B 0,C 180,E1 -12358.835,E2 -12358.835} C_VEL
LIN {X 0,Y 375.957,Z 159.152,A -85,B 0,C 180,E1 -12361.562,E2 -12361.562} C_VEL
LIN {X 0,Y 375.95,Z 159.153,A -85,B 0,C 180,E1 -12365.416,E2 -12365.416} C_VEL
LIN {X 0,Y 375.937,Z 159.155,A -85,B 0,C 180,E1 -12368.263,E2 -12368.263} C_VEL
LIN {X 0,Y 375.919,Z 159.155,A -85,B 0,C 180,E1 -12371.598,E2 -12371.598} C_VEL
LIN {X 0,Y 375.926,Z 159.159,A -85,B 0,C 180,E1 -12374.731,E2 -12374.731} C_VEL
LIN {X 0,Y 375.924,Z 159.161,A -85,B 0,C 180,E1 -12378.401,E2 -12378.401} C_VEL
LIN {X 0,Y 375.97,Z 159.15,A -85,B 0,C 180,E1 -12381.73,E2 -12381.73} C_VEL
LIN {X 0,Y 375.979,Z 159.148,A -85,B 0,C 180,E1 -12385.333,E2 -12385.333} C_VEL
LIN {X 0,Y 375.957,Z 159.154,A -85,B 0,C 180,E1 -12388.438,E2 -12388.438} C_VEL
LIN {X 0,Y 375.935,Z 159.159,A -85,B 0,C 180,E1 -12392.136,E2 -12392.136} C_VEL
LIN {X 0,Y 375.977,Z 159.152,A -85,B 0,C 180,E1 -12395.717,E2 -12395.717} C_VEL
LIN {X 0,Y 375.998,Z 159.146,A -85,B 0,C 180,E1 -12399.198,E2 -12399.198} C_VEL
LIN {X 0,Y 376.05,Z 159.139,A -85,B 0,C 180,E1 -12402.601,E2 -12402.601} C_VEL
LIN {X 0,Y 376.089,Z 159.135,A -85,B 0,C 180,E1 -12406.342,E2 -12406.342} C_VEL
LIN {X 0,Y 376.118,Z 159.131,A -85,B 0,C 180,E1 -12410.319,E2 -12410.319} C_VEL
LIN {X 0,Y 376.238,Z 159.121,A -85,B 0,C 180,E1 -12413.565,E2 -12413.565} C_VEL
LIN {X 0,Y 376.353,Z 159.103,A -85,B 0,C 180,E1 -12417.86,E2 -12417.86} C_VEL
LIN {X 0,Y 376.487,Z 159.085,A -85,B 0,C 180,E1 -12420,E2 -12420} C_VEL
LIN {X 0,Y 376.188,Z 159.128,A -85,B 0,C 180,E1 -12423.213,E2 -12423.213} C_VEL
LIN {X 0,Y 376.217,Z 159.119,A -85,B 0,C 180,E1 -12426.483,E2 -12426.483} C_VEL
LIN {X 0,Y 376.118,Z 159.131,A -85,B 0,C 180,E1 -12429.682,E2 -12429.682} C_VEL
LIN {X 0,Y 376.089,Z 159.134,A -85,B 0,C 180,E1 -12433.658,E2 -12433.658} C_VEL
LIN {X 0,Y 376.044,Z 159.14,A -85,B 0,C 180,E1 -12437.608,E2 -12437.608} C_VEL
LIN {X 0,Y 375.978,Z 159.152,A -85,B 0,C 180,E1 -12440.832,E2 -12440.832} C_VEL
LIN {X 0,Y 375.994,Z 159.15,A -85,B 0,C 180,E1 -12444.282,E2 -12444.282} C_VEL
LIN {X 0,Y 376.02,Z 159.147,A -85,B 0,C 180,E1 -12446.652,E2 -12446.652} C_VEL
LIN {X 0,Y 375.97,Z 159.149,A -85,B 0,C 180,E1 -12449.079,E2 -12449.079} C_VEL
LIN {X 0,Y 375.949,Z 159.153,A -85,B 0,C 180,E1 -12452.829,E2 -12452.829} C_VEL
LIN {X 0,Y 375.958,Z 159.151,A -85,B 0,C 180,E1 -12455.416,E2 -12455.416} C_VEL
LIN {X 0,Y 375.974,Z 159.153,A -85,B 0,C 180,E1 -12458.271,E2 -12458.271} C_VEL
LIN {X 0,Y 375.935,Z 159.156,A -85,B 0,C 180,E1 -12461.601,E2 -12461.601} C_VEL
LIN {X 0,Y 375.928,Z 159.155,A -85,B 0,C 180,E1 -12465.269,E2 -12465.269} C_VEL
LIN {X 0,Y 375.935,Z 159.154,A -85,B 0,C 180,E1 -12468.4,E2 -12468.4} C_VEL
LIN {X 0,Y 375.974,Z 159.155,A -85,B 0,C 180,E1 -12471.73,E2 -12471.73} C_VEL
LIN {X 0,Y 375.981,Z 159.151,A -85,B 0,C 180,E1 -12475.333,E2 -12475.333} C_VEL
LIN {X 0,Y 375.959,Z 159.15,A -85,B 0,C 180,E1 -12478.438,E2 -12478.438} C_VEL
LIN {X 0,Y 375.998,Z 159.15,A -85,B 0,C 180,E1 -12482.142,E2 -12482.142} C_VEL
LIN {X 0,Y 376.073,Z 159.261,A -85,B 0,C 180,E1 -12484.729,E2 -12484.729} C_VEL
LIN {X 0,Y 378.171,Z 170.019,A -85,B 0,C 180,E1 -12487.607,E2 -12487.607} C_VEL
LIN {X 0,Y 378.721,Z 174.813,A -85,B 0,C 180,E1 -12488.83,E2 -12488.83} C_VEL
LIN {X 0,Y 383.7,Z 199.111,A -85,B 0,C 180,E1 -12489.608,E2 -12489.608} C_VEL
LIN {X 0,Y 383.098,Z 249.419,A -85,B 0,C 180,E1 -12490.558,E2 -12490.558} C_VEL
LIN {X 0,Y 382.563,Z 282.789,A -85,B 0,C 180,E1 -12491.212,E2 -12491.212} C_VEL
LIN {X 0,Y 382.009,Z 296.604,A -85,B 0,C 180,E1 -12491.705,E2 -12491.705} C_VEL
LIN {X 0,Y 381.313,Z 308.981,A -85,B 0,C 180,E1 -12492.365,E2 -12492.365} C_VEL
LIN {X 0,Y 380.405,Z 320.824,A -85,B 0,C 180,E1 -12493.222,E2 -12493.222} C_VEL
LIN {X 0,Y 379.426,Z 332.575,A -85,B 0,C 180,E1 -12494.324,E2 -12494.324} C_VEL
LIN {X 0,Y 378.666,Z 342.421,A -85,B 0,C 180,E1 -12495.489,E2 -12495.489} C_VEL
LIN {X 0,Y 377.634,Z 351.61,A -85,B 0,C 180,E1 -12496.822,E2 -12496.822} C_VEL
LIN {X 0,Y 376.715,Z 360.531,A -85,B 0,C 180,E1 -12498.431,E2 -12498.431} C_VEL
LIN {X 0,Y 375.973,Z 367.712,A -85,B 0,C 180,E1 -12500.043,E2 -12500.043} C_VEL
LIN {X 0,Y 375.447,Z 372.556,A -85,B 0,C 180,E1 -12501.387,E2 -12501.387} C_VEL
LIN {X 0,Y 375.072,Z 377.263,A -85,B 0,C 180,E1 -12503.005,E2 -12503.005} C_VEL
LIN {X 0,Y 374.846,Z 380.862,A -85,B 0,C 180,E1 -12504.621,E2 -12504.621} C_VEL
LIN {X 0,Y 374.674,Z 382.725,A -85,B 0,C 180,E1 -12505.697,E2 -12505.697} C_VEL
LIN {X 0,Y 374.571,Z 384.127,A -85,B 0,C 180,E1 -12506.773,E2 -12506.773} C_VEL
LIN {X 0,Y 374.549,Z 385.123,A -85,B 0,C 180,E1 -12507.849,E2 -12507.849} C_VEL
LIN {X 0,Y 374.529,Z 385.736,A -85,B 0,C 180,E1 -12508.925,E2 -12508.925} C_VEL
LIN {X 0,Y 374.51,Z 385.97,A -85,B 0,C 180,E1 -12510,E2 -12510} C_VEL
LIN {X 0,Y 374.529,Z 385.78,A -85,B 0,C 180,E1 -12511.075,E2 -12511.075} C_VEL
LIN {X 0,Y 374.548,Z 385.196,A -85,B 0,C 180,E1 -12512.151,E2 -12512.151} C_VEL
LIN {X 0,Y 374.667,Z 382.871,A -85,B 0,C 180,E1 -12514.303,E2 -12514.303} C_VEL
LIN {X 0,Y 374.912,Z 380.002,A -85,B 0,C 180,E1 -12515.918,E2 -12515.918} C_VEL
LIN {X 0,Y 375.157,Z 376.113,A -85,B 0,C 180,E1 -12517.535,E2 -12517.535} C_VEL
LIN {X 0,Y 375.616,Z 371.094,A -85,B 0,C 180,E1 -12519.151,E2 -12519.151} C_VEL
LIN {X 0,Y 376.275,Z 364.775,A -85,B 0,C 180,E1 -12520.765,E2 -12520.765} C_VEL
LIN {X 0,Y 377.06,Z 356.866,A -85,B 0,C 180,E1 -12522.377,E2 -12522.377} C_VEL
LIN {X 0,Y 377.851,Z 350.394,A -85,B 0,C 180,E1 -12523.472,E2 -12523.472} C_VEL
LIN {X 0,Y 377.621,Z 346.285,A -85,B 0,C 180,E1 -12524.112,E2 -12524.112} C_VEL
LIN {X 0,Y 375.43,Z 339.374,A -85,B 0,C 180,E1 -12525.15,E2 -12525.15} C_VEL
LIN {X 0,Y 373.303,Z 332.06,A -85,B 0,C 180,E1 -12526.12,E2 -12526.12} C_VEL
LIN {X 0,Y 373.142,Z 327.21,A -85,B 0,C 180,E1 -12526.634,E2 -12526.634} C_VEL
LIN {X 0,Y 374.123,Z 315.431,A -85,B 0,C 180,E1 -12527.632,E2 -12527.632} C_VEL
LIN {X 0,Y 375.022,Z 302.823,A -85,B 0,C 180,E1 -12528.436,E2 -12528.436} C_VEL
LIN {X 0,Y 375.623,Z 289.273,A -85,B 0,C 180,E1 -12529.042,E2 -12529.042} C_VEL
LIN {X 0,Y 376.064,Z 277.213,A -85,B 0,C 180,E1 -12529.373,E2 -12529.373} C_VEL
LIN {X 0,Y 377.142,Z 200.559,A -85,B 0,C 180,E1 -12530.841,E2 -12530.841} C_VEL
LIN {X 0,Y 372.169,Z 176.471,A -85,B 0,C 180,E1 -12531.625,E2 -12531.625} C_VEL
LIN {X 0,Y 371.816,Z 174.863,A -85,B 0,C 180,E1 -12531.718,E2 -12531.718} C_VEL
LIN {X 0,Y 370.095,Z 165.267,A -85,B 0,C 180,E1 -12534.285,E2 -12534.285} C_VEL
LIN {X 0,Y 369.012,Z 160.019,A -85,B 0,C 180,E1 -12535.752,E2 -12535.752} C_VEL
LIN {X 0,Y 368.963,Z 160.027,A -85,B 0,C 180,E1 -12538.811,E2 -12538.811} C_VEL
LIN {X 0,Y 368.899,Z 160.033,A -85,B 0,C 180,E1 -12542.238,E2 -12542.238} C_VEL
LIN {X 0,Y 368.93,Z 160.028,A -85,B 0,C 180,E1 -12545.001,E2 -12545.001} C_VEL
LIN {X 0,Y 368.908,Z 160.032,A -85,B 0,C 180,E1 -12548.64,E2 -12548.64} C_VEL
LIN {X 0,Y 368.882,Z 160.035,A -85,B 0,C 180,E1 -12552.009,E2 -12552.009} C_VEL
LIN {X 0,Y 368.881,Z 160.032,A -85,B 0,C 180,E1 -12555.176,E2 -12555.176} C_VEL
LIN {X 0,Y 368.883,Z 160.037,A -85,B 0,C 180,E1 -12558.177,E2 -12558.177} C_VEL
LIN {X 0,Y 368.908,Z 160.03,A -85,B 0,C 180,E1 -12561.36,E2 -12561.36} C_VEL
LIN {X 0,Y 368.936,Z 160.026,A -85,B 0,C 180,E1 -12565.146,E2 -12565.146} C_VEL
LIN {X 0,Y 368.929,Z 160.027,A -85,B 0,C 180,E1 -12569.046,E2 -12569.046} C_VEL
LIN {X 0,Y 368.979,Z 160.025,A -85,B 0,C 180,E1 -12571.564,E2 -12571.564} C_VEL
LIN {X 0,Y 369,Z 160.02,A -85,B 0,C 180,E1 -12574.02,E2 -12574.02} C_VEL
LIN {X 0,Y 368.932,Z 160.031,A -85,B 0,C 180,E1 -12577.605,E2 -12577.605} C_VEL
LIN {X 0,Y 368.982,Z 160.023,A -85,B 0,C 180,E1 -12581.107,E2 -12581.107} C_VEL
LIN {X 0,Y 368.997,Z 160.018,A -85,B 0,C 180,E1 -12584.535,E2 -12584.535} C_VEL
LIN {X 0,Y 369.004,Z 160.017,A -85,B 0,C 180,E1 -12587.907,E2 -12587.907} C_VEL
LIN {X 0,Y 369.186,Z 159.994,A -85,B 0,C 180,E1 -12591.846,E2 -12591.846} C_VEL
LIN {X 0,Y 369.141,Z 160.002,A -85,B 0,C 180,E1 -12594.537,E2 -12594.537} C_VEL
LIN {X 0,Y 369.318,Z 159.978,A -85,B 0,C 180,E1 -12597.819,E2 -12597.819} C_VEL
LIN {X 0,Y 369.456,Z 159.961,A -85,B 0,C 180,E1 -12600,E2 -12600} C_VEL
LIN {X 0,Y 369.317,Z 159.979,A -85,B 0,C 180,E1 -12602.181,E2 -12602.181} C_VEL
LIN {X 0,Y 369.198,Z 159.999,A -85,B 0,C 180,E1 -12606.558,E2 -12606.558} C_VEL
LIN {X 0,Y 369.12,Z 160.006,A -85,B 0,C 180,E1 -12608.761,E2 -12608.761} C_VEL
LIN {X 0,Y 369.004,Z 160.02,A -85,B 0,C 180,E1 -12612.093,E2 -12612.093} C_VEL
LIN {X 0,Y 368.997,Z 160.018,A -85,B 0,C 180,E1 -12615.465,E2 -12615.465} C_VEL
LIN {X 0,Y 368.965,Z 160.022,A -85,B 0,C 180,E1 -12618.894,E2 -12618.894} C_VEL
LIN {X 0,Y 368.921,Z 160.031,A -85,B 0,C 180,E1 -12622.396,E2 -12622.396} C_VEL
LIN {X 0,Y 368.999,Z 160.023,A -85,B 0,C 180,E1 -12625.98,E2 -12625.98} C_VEL
LIN {X 0,Y 368.914,Z 160.032,A -85,B 0,C 180,E1 -12629.69,E2 -12629.69} C_VEL
LIN {X 0,Y 368.896,Z 160.031,A -85,B 0,C 180,E1 -12633.043,E2 -12633.043} C_VEL
LIN {X 0,Y 368.916,Z 160.03,A -85,B 0,C 180,E1 -12636.197,E2 -12636.197} C_VEL
LIN {X 0,Y 368.895,Z 160.031,A -85,B 0,C 180,E1 -12638.954,E2 -12638.954} C_VEL
LIN {X 0,Y 368.874,Z 160.035,A -85,B 0,C 180,E1 -12642.008,E2 -12642.008} C_VEL
LIN {X 0,Y 368.879,Z 160.036,A -85,B 0,C 180,E1 -12645.176,E2 -12645.176} C_VEL
LIN {X 0,Y 368.87,Z 160.034,A -85,B 0,C 180,E1 -12648.176,E2 -12648.176} C_VEL
LIN {X 0,Y 368.878,Z 160.038,A -85,B 0,C 180,E1 -12651.366,E2 -12651.366} C_VEL
LIN {X 0,Y 368.937,Z 160.032,A -85,B 0,C 180,E1 -12655.147,E2 -12655.147} C_VEL
LIN {X 0,Y 368.93,Z 160.032,A -85,B 0,C 180,E1 -12659.047,E2 -12659.047} C_VEL
LIN {X 0,Y 368.95,Z 160.109,A -85,B 0,C 180,E1 -12660.848,E2 -12660.848} C_VEL
LIN {X 0,Y 371.404,Z 171.806,A -85,B 0,C 180,E1 -12663.899,E2 -12663.899} C_VEL
LIN {X 0,Y 372.534,Z 179.333,A -85,B 0,C 180,E1 -12665.775,E2 -12665.775} C_VEL
LIN {X 0,Y 371.518,Z 190.417,A -85,B 0,C 180,E1 -12668.325,E2 -12668.325} C_VEL
LIN {X 0,Y 376.526,Z 219.683,A -85,B 0,C 180,E1 -12669.229,E2 -12669.229} C_VEL
LIN {X 0,Y 376.856,Z 225.579,A -85,B 0,C 180,E1 -12669.365,E2 -12669.365} C_VEL
LIN {X 0,Y 375.692,Z 298.794,A -85,B 0,C 180,E1 -12670.785,E2 -12670.785} C_VEL
LIN {X 0,Y 375.036,Z 311.999,A -85,B 0,C 180,E1 -12671.246,E2 -12671.246} C_VEL
LIN {X 0,Y 374.282,Z 324.126,A -85,B 0,C 180,E1 -12671.881,E2 -12671.881} C_VEL
LIN {X 0,Y 373.259,Z 336.363,A -85,B 0,C 180,E1 -12672.749,E2 -12672.749} C_VEL
LIN {X 0,Y 372.124,Z 347.941,A -85,B 0,C 180,E1 -12673.825,E2 -12673.825} C_VEL
LIN {X 0,Y 371.142,Z 358.595,A -85,B 0,C 180,E1 -12675.078,E2 -12675.078} C_VEL
LIN {X 0,Y 370.326,Z 366.897,A -85,B 0,C 180,E1 -12676.277,E2 -12676.277} C_VEL
LIN {X 0,Y 369.449,Z 374.763,A -85,B 0,C 180,E1 -12677.643,E2 -12677.643} C_VEL
LIN {X 0,Y 368.65,Z 382.446,A -85,B 0,C 180,E1 -12679.288,E2 -12679.288} C_VEL
LIN {X 0,Y 367.999,Z 389.533,A -85,B 0,C 180,E1 -12681.212,E2 -12681.212} C_VEL
LIN {X 0,Y 367.661,Z 394.248,A -85,B 0,C 180,E1 -12682.863,E2 -12682.863} C_VEL
LIN {X 0,Y 367.462,Z 397.851,A -85,B 0,C 180,E1 -12684.513,E2 -12684.513} C_VEL
LIN {X 0,Y 367.43,Z 399.71,A -85,B 0,C 180,E1 -12685.612,E2 -12685.612} C_VEL
LIN {X 0,Y 367.369,Z 401.103,A -85,B 0,C 180,E1 -12686.71,E2 -12686.71} C_VEL
LIN {X 0,Y 367.389,Z 402.705,A -85,B 0,C 180,E1 -12688.904,E2 -12688.904} C_VEL
LIN {X 0,Y 367.41,Z 402.919,A -85,B 0,C 180,E1 -12690,E2 -12690} C_VEL
LIN {X 0,Y 367.389,Z 402.7,A -85,B 0,C 180,E1 -12691.096,E2 -12691.096} C_VEL
LIN {X 0,Y 367.369,Z 401.094,A -85,B 0,C 180,E1 -12693.29,E2 -12693.29} C_VEL
LIN {X 0,Y 367.43,Z 399.696,A -85,B 0,C 180,E1 -12694.388,E2 -12694.388} C_VEL
LIN {X 0,Y 367.479,Z 396.806,A -85,B 0,C 180,E1 -12696.013,E2 -12696.013} C_VEL
LIN {X 0,Y 367.722,Z 392.783,A -85,B 0,C 180,E1 -12697.688,E2 -12697.688} C_VEL
LIN {X 0,Y 368.215,Z 386.672,A -85,B 0,C 180,E1 -12699.614,E2 -12699.614} C_VEL
LIN {X 0,Y 368.841,Z 379.996,A -85,B 0,C 180,E1 -12701.263,E2 -12701.263} C_VEL
LIN {X 0,Y 369.772,Z 371.717,A -85,B 0,C 180,E1 -12702.904,E2 -12702.904} C_VEL
LIN {X 0,Y 370.6,Z 363.226,A -85,B 0,C 180,E1 -12704.272,E2 -12704.272} C_VEL
LIN {X 0,Y 371.637,Z 352.735,A -85,B 0,C 180,E1 -12705.633,E2 -12705.633} C_VEL
LIN {X 0,Y 372.803,Z 340.928,A -85,B 0,C 180,E1 -12706.849,E2 -12706.849} C_VEL
LIN {X 0,Y 373.843,Z 329.045,A -85,B 0,C 180,E1 -12707.788,E2 -12707.788} C_VEL
LIN {X 0,Y 374.698,Z 316.677,A -85,B 0,C 180,E1 -12708.523,E2 -12708.523} C_VEL
LIN {X 0,Y 375.454,Z 303.964,A -85,B 0,C 180,E1 -12709.051,E2 -12709.051} C_VEL
LIN {X 0,Y 375.903,Z 290.587,A -85,B 0,C 180,E1 -12709.382,E2 -12709.382} C_VEL
LIN {X 0,Y 376.753,Z 221.206,A -85,B 0,C 180,E1 -12710.714,E2 -12710.714} C_VEL
LIN {X 0,Y 371.516,Z 190.479,A -85,B 0,C 180,E1 -12711.646,E2 -12711.646} C_VEL
LIN {X 0,Y 372.544,Z 179.266,A -85,B 0,C 180,E1 -12714.224,E2 -12714.224} C_VEL
LIN {X 0,Y 371.607,Z 172.993,A -85,B 0,C 180,E1 -12715.784,E2 -12715.784} C_VEL
LIN {X 0,Y 369.504,Z 162.925,A -85,B 0,C 180,E1 -12718.392,E2 -12718.392} C_VEL
LIN {X 0,Y 368.892,Z 160.035,A -85,B 0,C 180,E1 -12719.192,E2 -12719.192} C_VEL
LIN {X 0,Y 368.897,Z 160.031,A -85,B 0,C 180,E1 -12722.238,E2 -12722.238} C_VEL
LIN {X 0,Y 368.924,Z 160.032,A -85,B 0,C 180,E1 -12725,E2 -12725} C_VEL
LIN {X 0,Y 368.878,Z 160.037,A -85,B 0,C 180,E1 -12728.634,E2 -12728.634} C_VEL
LIN {X 0,Y 368.871,Z 160.034,A -85,B 0,C 180,E1 -12732.007,E2 -12732.007} C_VEL
LIN {X 0,Y 368.879,Z 160.033,A -85,B 0,C 180,E1 -12735.176,E2 -12735.176} C_VEL
LIN {X 0,Y 368.874,Z 160.036,A -85,B 0,C 180,E1 -12738.176,E2 -12738.176} C_VEL
LIN {X 0,Y 368.902,Z 160.029,A -85,B 0,C 180,E1 -12741.361,E2 -12741.361} C_VEL
LIN {X 0,Y 368.936,Z 160.025,A -85,B 0,C 180,E1 -12745.146,E2 -12745.146} C_VEL
LIN {X 0,Y 368.929,Z 160.026,A -85,B 0,C 180,E1 -12749.046,E2 -12749.046} C_VEL
LIN {X 0,Y 368.878,Z 160.033,A -85,B 0,C 180,E1 -12752.79,E2 -12752.79} C_VEL
LIN {X 0,Y 368.928,Z 160.031,A -85,B 0,C 180,E1 -12756.119,E2 -12756.119} C_VEL
LIN {X 0,Y 368.936,Z 160.03,A -85,B 0,C 180,E1 -12759.947,E2 -12759.947} C_VEL
LIN {X 0,Y 368.976,Z 160.023,A -85,B 0,C 180,E1 -12763.399,E2 -12763.399} C_VEL
LIN {X 0,Y 369.057,Z 160.01,A -85,B 0,C 180,E1 -12766.79,E2 -12766.79} C_VEL
LIN {X 0,Y 369.067,Z 160.01,A -85,B 0,C 180,E1 -12770.132,E2 -12770.132} C_VEL
LIN {X 0,Y 369.198,Z 159.999,A -85,B 0,C 180,E1 -12773.442,E2 -12773.442} C_VEL
LIN {X 0,Y 369.318,Z 159.979,A -85,B 0,C 180,E1 -12777.819,E2 -12777.819} C_VEL
LIN {X 0,Y 369.456,Z 159.961,A -85,B 0,C 180,E1 -12780,E2 -12780} C_VEL
LIN {X 0,Y 369.319,Z 159.978,A -85,B 0,C 180,E1 -12782.181,E2 -12782.181} C_VEL
LIN {X 0,Y 369.183,Z 159.996,A -85,B 0,C 180,E1 -12786.559,E2 -12786.559} C_VEL
LIN {X 0,Y 369.106,Z 160.008,A -85,B 0,C 180,E1 -12788.762,E2 -12788.762} C_VEL
LIN {X 0,Y 369.004,Z 160.017,A -85,B 0,C 180,E1 -12792.093,E2 -12792.093} C_VEL
LIN {X 0,Y 368.998,Z 160.018,A -85,B 0,C 180,E1 -12795.465,E2 -12795.465} C_VEL
LIN {X 0,Y 368.983,Z 160.023,A -85,B 0,C 180,E1 -12798.893,E2 -12798.893} C_VEL
LIN {X 0,Y 368.933,Z 160.03,A -85,B 0,C 180,E1 -12802.395,E2 -12802.395} C_VEL
LIN {X 0,Y 369,Z 160.019,A -85,B 0,C 180,E1 -12805.98,E2 -12805.98} C_VEL
LIN {X 0,Y 368.961,Z 160.024,A -85,B 0,C 180,E1 -12808.812,E2 -12808.812} C_VEL
LIN {X 0,Y 368.898,Z 160.036,A -85,B 0,C 180,E1 -12812.238,E2 -12812.238} C_VEL
LIN {X 0,Y 368.929,Z 160.026,A -85,B 0,C 180,E1 -12815.002,E2 -12815.002} C_VEL
LIN {X 0,Y 368.908,Z 160.03,A -85,B 0,C 180,E1 -12818.64,E2 -12818.64} C_VEL
LIN {X 0,Y 368.883,Z 160.038,A -85,B 0,C 180,E1 -12822.01,E2 -12822.01} C_VEL
LIN {X 0,Y 368.881,Z 160.033,A -85,B 0,C 180,E1 -12825.176,E2 -12825.176} C_VEL
LIN {X 0,Y 368.884,Z 160.034,A -85,B 0,C 180,E1 -12828.178,E2 -12828.178} C_VEL
LIN {X 0,Y 368.908,Z 160.032,A -85,B 0,C 180,E1 -12831.36,E2 -12831.36} C_VEL
LIN {X 0,Y 368.938,Z 160.027,A -85,B 0,C 180,E1 -12835.147,E2 -12835.147} C_VEL
LIN {X 0,Y 368.931,Z 160.028,A -85,B 0,C 180,E1 -12839.047,E2 -12839.047} C_VEL
LIN {X 0,Y 368.982,Z 160.025,A -85,B 0,C 180,E1 -12841.564,E2 -12841.564} C_VEL
LIN {X 0,Y 369.015,Z 160.131,A -85,B 0,C 180,E1 -12844.4,E2 -12844.4} C_VEL
LIN {X 0,Y 371.233,Z 171.333,A -85,B 0,C 180,E1 -12847.458,E2 -12847.458} C_VEL
LIN {X 0,Y 371.861,Z 175.285,A -85,B 0,C 180,E1 -12848.438,E2 -12848.438} C_VEL
LIN {X 0,Y 376.947,Z 199.463,A -85,B 0,C 180,E1 -12849.23,E2 -12849.23} C_VEL
LIN {X 0,Y 377.121,Z 206.417,A -85,B 0,C 180,E1 -12849.379,E2 -12849.379} C_VEL
LIN {X 0,Y 375.896,Z 281.789,A -85,B 0,C 180,E1 -12850.831,E2 -12850.831} C_VEL
LIN {X 0,Y 375.377,Z 295.255,A -85,B 0,C 180,E1 -12851.299,E2 -12851.299} C_VEL
LIN {X 0,Y 374.622,Z 308.049,A -85,B 0,C 180,E1 -12851.968,E2 -12851.968} C_VEL
LIN {X 0,Y 373.78,Z 319.404,A -85,B 0,C 180,E1 -12852.774,E2 -12852.774} C_VEL
LIN {X 0,Y 372.779,Z 330.809,A -85,B 0,C 180,E1 -12853.826,E2 -12853.826} C_VEL
LIN {X 0,Y 372.004,Z 340.461,A -85,B 0,C 180,E1 -12854.944,E2 -12854.944} C_VEL
LIN {X 0,Y 370.963,Z 350.078,A -85,B 0,C 180,E1 -12856.301,E2 -12856.301} C_VEL
LIN {X 0,Y 370.052,Z 357.956,A -85,B 0,C 180,E1 -12857.663,E2 -12857.663} C_VEL
LIN {X 0,Y 369.201,Z 365.655,A -85,B 0,C 180,E1 -12859.304,E2 -12859.304} C_VEL
LIN {X 0,Y 368.411,Z 372.721,A -85,B 0,C 180,E1 -12861.222,E2 -12861.222} C_VEL
LIN {X 0,Y 368.015,Z 377.426,A -85,B 0,C 180,E1 -12862.87,E2 -12862.87} C_VEL
LIN {X 0,Y 367.778,Z 381.026,A -85,B 0,C 180,E1 -12864.517,E2 -12864.517} C_VEL
LIN {X 0,Y 367.608,Z 382.888,A -85,B 0,C 180,E1 -12865.614,E2 -12865.614} C_VEL
LIN {X 0,Y 367.485,Z 384.289,A -85,B 0,C 180,E1 -12866.711,E2 -12866.711} C_VEL
LIN {X 0,Y 367.431,Z 385.898,A -85,B 0,C 180,E1 -12868.904,E2 -12868.904} C_VEL
LIN {X 0,Y 367.412,Z 386.132,A -85,B 0,C 180,E1 -12870,E2 -12870} C_VEL
LIN {X 0,Y 367.431,Z 385.942,A -85,B 0,C 180,E1 -12871.096,E2 -12871.096} C_VEL
LIN {X 0,Y 367.483,Z 384.391,A -85,B 0,C 180,E1 -12873.289,E2 -12873.289} C_VEL
LIN {X 0,Y 367.6,Z 383.033,A -85,B 0,C 180,E1 -12874.386,E2 -12874.386} C_VEL
LIN {X 0,Y 367.84,Z 379.848,A -85,B 0,C 180,E1 -12876.189,E2 -12876.189} C_VEL
LIN {X 0,Y 368.109,Z 376.274,A -85,B 0,C 180,E1 -12877.68,E2 -12877.68} C_VEL
LIN {X 0,Y 368.587,Z 371.255,A -85,B 0,C 180,E1 -12879.327,E2 -12879.327} C_VEL
LIN {X 0,Y 369.279,Z 364.936,A -85,B 0,C 180,E1 -12880.971,E2 -12880.971} C_VEL
LIN {X 0,Y 370.132,Z 357.025,A -85,B 0,C 180,E1 -12882.613,E2 -12882.613} C_VEL
LIN {X 0,Y 371.125,Z 348.958,A -85,B 0,C 180,E1 -12883.972,E2 -12883.972} C_VEL
LIN {X 0,Y 372.06,Z 339.118,A -85,B 0,C 180,E1 -12885.334,E2 -12885.334} C_VEL
LIN {X 0,Y 373.054,Z 328.049,A -85,B 0,C 180,E1 -12886.555,E2 -12886.555} C_VEL
LIN {X 0,Y 373.142,Z 327.21,A -85,B 0,C 180,E1 -12886.634,E2 -12886.634} C_VEL
LIN {X 0,Y 373.045,Z 322.237,A -85,B 0,C 180,E1 -12887.115,E2 -12887.115} C_VEL
LIN {X 0,Y 371.101,Z 313.949,A -85,B 0,C 180,E1 -12887.903,E2 -12887.903} C_VEL
LIN {X 0,Y 368.929,Z 305.402,A -85,B 0,C 180,E1 -12888.604,E2 -12888.604} C_VEL
LIN {X 0,Y 368.49,Z 299.934,A -85,B 0,C 180,E1 -12888.944,E2 -12888.944} C_VEL
LIN {X 0,Y 369.021,Z 287.564,A -85,B 0,C 180,E1 -12889.468,E2 -12889.468} C_VEL
LIN {X 0,Y 369.47,Z 273.909,A -85,B 0,C 180,E1 -12889.805,E2 -12889.805} C_VEL
LIN {X 0,Y 370.475,Z 201.397,A -85,B 0,C 180,E1 -12891.22,E2 -12891.22} C_VEL
LIN {X 0,Y 365.847,Z 178.737,A -85,B 0,C 180,E1 -12891.973,E2 -12891.973} C_VEL
LIN {X 0,Y 364.741,Z 175.155,A -85,B 0,C 180,E1 -12892.129,E2 -12892.129} C_VEL
LIN {X 0,Y 362.604,Z 163.853,A -85,B 0,C 180,E1 -12895.239,E2 -12895.239} C_VEL
LIN {X 0,Y 361.96,Z 160.897,A -85,B 0,C 180,E1 -12896.136,E2 -12896.136} C_VEL
LIN {X 0,Y 361.914,Z 160.902,A -85,B 0,C 180,E1 -12899.09,E2 -12899.09} C_VEL
LIN {X 0,Y 361.85,Z 160.911,A -85,B 0,C 180,E1 -12902.944,E2 -12902.944} C_VEL
LIN {X 0,Y 361.869,Z 160.906,A -85,B 0,C 180,E1 -12905.636,E2 -12905.636} C_VEL
LIN {X 0,Y 361.869,Z 160.906,A -85,B 0,C 180,E1 -12909.026,E2 -12909.026} C_VEL
LIN {X 0,Y 361.837,Z 160.911,A -85,B 0,C 180,E1 -12912.828,E2 -12912.828} C_VEL
LIN {X 0,Y 361.819,Z 160.916,A -85,B 0,C 180,E1 -12915.946,E2 -12915.946} C_VEL
LIN {X 0,Y 361.835,Z 160.91,A -85,B 0,C 180,E1 -12919.244,E2 -12919.244} C_VEL
LIN {X 0,Y 361.863,Z 160.906,A -85,B 0,C 180,E1 -12922.777,E2 -12922.777} C_VEL
LIN {X 0,Y 361.854,Z 160.912,A -85,B 0,C 180,E1 -12925.719,E2 -12925.719} C_VEL
LIN {X 0,Y 361.874,Z 160.911,A -85,B 0,C 180,E1 -12929.672,E2 -12929.672} C_VEL
LIN {X 0,Y 361.954,Z 160.899,A -85,B 0,C 180,E1 -12933.475,E2 -12933.475} C_VEL
LIN {X 0,Y 361.89,Z 160.906,A -85,B 0,C 180,E1 -12937.145,E2 -12937.145} C_VEL
LIN {X 0,Y 361.92,Z 160.9,A -85,B 0,C 180,E1 -12940.724,E2 -12940.724} C_VEL
LIN {X 0,Y 361.945,Z 160.896,A -85,B 0,C 180,E1 -12944.226,E2 -12944.226} C_VEL
